LIN {X 0,Y 322.376,Z 758.442,A -85,B 0,C 180,E1 13709.907,E2 13709.907} C_VEL
LIN {X 0,Y 327.986,Z 742.44,A -85,B 0,C 180,E1 13707.682,E2 13707.682} C_VEL
LIN {X 0,Y 333.329,Z 725.588,A -85,B 0,C 180,E1 13705.781,E2 13705.781} C_VEL
LIN {X 0,Y 338.292,Z 707.747,A -85,B 0,C 180,E1 13704.157,E2 13704.157} C_VEL
LIN {X 0,Y 342.895,Z 688.344,A -85,B 0,C 180,E1 13702.762,E2 13702.762} C_VEL
LIN {X 0,Y 346.893,Z 667.6,A -85,B 0,C 180,E1 13701.623,E2 13701.623} C_VEL
LIN {X 0,Y 350,Z 646.538,A -85,B 0,C 180,E1 13700.791,E2 13700.791} C_VEL
LIN {X 0,Y 352.547,Z 620.24,A -85,B 0,C 180,E1 13700.102,E2 13700.102} C_VEL
LIN {X 0,Y 365.107,Z 463.823,A -85,B 0,C 180,E1 13696.583,E2 13696.583} C_VEL
LIN {X 0,Y 364.004,Z 412.304,A -85,B 0,C 180,E1 13693.947,E2 13693.947} C_VEL
LIN {X 0,Y 363.272,Z 382.468,A -85,B 0,C 180,E1 13692.235,E2 13692.235} C_VEL
LIN {X 0,Y 360.522,Z 376.636,A -85,B 0,C 180,E1 13690.87,E2 13690.87} C_VEL
LIN {X 0,Y 357.367,Z 367.476,A -85,B 0,C 180,E1 13688.041,E2 13688.041} C_VEL
LIN {X 0,Y 354.327,Z 359.067,A -85,B 0,C 180,E1 13684.856,E2 13684.856} C_VEL
LIN {X 0,Y 352.321,Z 354.194,A -85,B 0,C 180,E1 13682.439,E2 13682.439} C_VEL
LIN {X 0,Y 351.131,Z 351.132,A -85,B 0,C 180,E1 13680.652,E2 13680.652} C_VEL
LIN {X 0,Y 350.069,Z 347.943,A -85,B 0,C 180,E1 13678.363,E2 13678.363} C_VEL
LIN {X 0,Y 348.93,Z 344.03,A -85,B 0,C 180,E1 13673.583,E2 13673.583} C_VEL
LIN {X 0,Y 349.355,Z 344.256,A -85,B 0,C 180,E1 13668.944,E2 13668.944} C_VEL
LIN {X 0,Y 351.588,Z 349.237,A -85,B 0,C 180,E1 13663.817,E2 13663.817} C_VEL
LIN {X 0,Y 353.437,Z 352.672,A -85,B 0,C 180,E1 13661.698,E2 13661.698} C_VEL
LIN {X 0,Y 358.022,Z 358.691,A -85,B 0,C 180,E1 13659.226,E2 13659.226} C_VEL
LIN {X 0,Y 362.84,Z 365.211,A -85,B 0,C 180,E1 13657.05,E2 13657.05} C_VEL
LIN {X 0,Y 369.826,Z 375.683,A -85,B 0,C 180,E1 13654.369,E2 13654.369} C_VEL
LIN {X 0,Y 374.027,Z 382.841,A -85,B 0,C 180,E1 13652.929,E2 13652.929} C_VEL
LIN {X 0,Y 364.112,Z 552.249,A -85,B 0,C 180,E1 13649.475,E2 13649.475} C_VEL
LIN {X 0,Y 358.709,Z 656.095,A -85,B 0,C 180,E1 13647.399,E2 13647.399} C_VEL
LIN {X 0,Y 356.14,Z 678.482,A -85,B 0,C 180,E1 13646.754,E2 13646.754} C_VEL
LIN {X 0,Y 352.594,Z 700.34,A -85,B 0,C 180,E1 13645.893,E2 13645.893} C_VEL
LIN {X 0,Y 348.351,Z 721.516,A -85,B 0,C 180,E1 13644.793,E2 13644.793} C_VEL
LIN {X 0,Y 343.457,Z 741.511,A -85,B 0,C 180,E1 13643.46,E2 13643.46} C_VEL
LIN {X 0,Y 337.812,Z 761.919,A -85,B 0,C 180,E1 13641.786,E2 13641.786} C_VEL
LIN {X 0,Y 331.997,Z 780.753,A -85,B 0,C 180,E1 13639.9,E2 13639.9} C_VEL
LIN {X 0,Y 325.618,Z 799.71,A -85,B 0,C 180,E1 13637.599,E2 13637.599} C_VEL
LIN {X 0,Y 319.339,Z 817.406,A -85,B 0,C 180,E1 13635.038,E2 13635.038} C_VEL
LIN {X 0,Y 313.159,Z 834.22,A -85,B 0,C 180,E1 13632.102,E2 13632.102} C_VEL
LIN {X 0,Y 307.081,Z 850.603,A -85,B 0,C 180,E1 13628.69,E2 13628.69} C_VEL
LIN {X 0,Y 301.905,Z 865.076,A -85,B 0,C 180,E1 13625.112,E2 13625.112} C_VEL
LIN {X 0,Y 297.411,Z 878.3,A -85,B 0,C 180,E1 13621.177,E2 13621.177} C_VEL
LIN {X 0,Y 293.801,Z 890.287,A -85,B 0,C 180,E1 13616.909,E2 13616.909} C_VEL
LIN {X 0,Y 291.315,Z 900.346,A -85,B 0,C 180,E1 13612.605,E2 13612.605} C_VEL
LIN {X 0,Y 289.82,Z 908.415,A -85,B 0,C 180,E1 13608.295,E2 13608.295} C_VEL
LIN {X 0,Y 289.1,Z 914.862,A -85,B 0,C 180,E1 13604.008,E2 13604.008} C_VEL
LIN {X 0,Y 288.923,Z 919.155,A -85,B 0,C 180,E1 13600.163,E2 13600.163} C_VEL
LIN {X 0,Y 289.025,Z 922.186,A -85,B 0,C 180,E1 13596.354,E2 13596.354} C_VEL
LIN {X 0,Y 289.148,Z 923.885,A -85,B 0,C 180,E1 13592.376,E2 13592.376} C_VEL
LIN {X 0,Y 289.163,Z 924.136,A -85,B 0,C 180,E1 13589.007,E2 13589.007} C_VEL
LIN {X 0,Y 289.07,Z 923.328,A -85,B 0,C 180,E1 13585.634,E2 13585.634} C_VEL
LIN {X 0,Y 288.916,Z 921.176,A -85,B 0,C 180,E1 13581.798,E2 13581.798} C_VEL
LIN {X 0,Y 288.954,Z 917.176,A -85,B 0,C 180,E1 13577.61,E2 13577.61} C_VEL
LIN {X 0,Y 289.353,Z 912.158,A -85,B 0,C 180,E1 13573.744,E2 13573.744} C_VEL
LIN {X 0,Y 290.48,Z 904.897,A -85,B 0,C 180,E1 13569.432,E2 13569.432} C_VEL
LIN {X 0,Y 292.375,Z 896.411,A -85,B 0,C 180,E1 13565.339,E2 13565.339} C_VEL
LIN {X 0,Y 295.239,Z 886.029,A -85,B 0,C 180,E1 13561.254,E2 13561.254} C_VEL
LIN {X 0,Y 298.941,Z 874.449,A -85,B 0,C 180,E1 13557.417,E2 13557.417} C_VEL
LIN {X 0,Y 303.355,Z 861.486,A -85,B 0,C 180,E1 13553.842,E2 13553.842} C_VEL
LIN {X 0,Y 309.063,Z 845.63,A -85,B 0,C 180,E1 13550.165,E2 13550.165} C_VEL
LIN {X 0,Y 314.851,Z 829.645,A -85,B 0,C 180,E1 13547.062,E2 13547.062} C_VEL
LIN {X 0,Y 320.804,Z 812.678,A -85,B 0,C 180,E1 13544.331,E2 13544.331} C_VEL
LIN {X 0,Y 327.159,Z 793.761,A -85,B 0,C 180,E1 13541.778,E2 13541.778} C_VEL
LIN {X 0,Y 333.113,Z 774.835,A -85,B 0,C 180,E1 13539.653,E2 13539.653} C_VEL
LIN {X 0,Y 338.667,Z 754.972,A -85,B 0,C 180,E1 13537.836,E2 13537.836} C_VEL
LIN {X 0,Y 344.127,Z 733.064,A -85,B 0,C 180,E1 13536.208,E2 13536.208} C_VEL
LIN {X 0,Y 348.613,Z 712.087,A -85,B 0,C 180,E1 13534.964,E2 13534.964} C_VEL
LIN {X 0,Y 352.338,Z 690.211,A -85,B 0,C 180,E1 13533.974,E2 13533.974} C_VEL
LIN {X 0,Y 355.448,Z 666.338,A -85,B 0,C 180,E1 13533.189,E2 13533.189} C_VEL
LIN {X 0,Y 357.156,Z 643.717,A -85,B 0,C 180,E1 13532.651,E2 13532.651} C_VEL
LIN {X 0,Y 366.358,Z 456.176,A -85,B 0,C 180,E1 13528.938,E2 13528.938} C_VEL
LIN {X 0,Y 370.274,Z 382.007,A -85,B 0,C 180,E1 13527.414,E2 13527.414} C_VEL
LIN {X 0,Y 359.115,Z 365.438,A -85,B 0,C 180,E1 13524.51,E2 13524.51} C_VEL
LIN {X 0,Y 349.693,Z 352.331,A -85,B 0,C 180,E1 13521.821,E2 13521.821} C_VEL
LIN {X 0,Y 340.937,Z 340.666,A -85,B 0,C 180,E1 13518.998,E2 13518.998} C_VEL
LIN {X 0,Y 335.21,Z 330.431,A -85,B 0,C 180,E1 13515.573,E2 13515.573} C_VEL
LIN {X 0,Y 329.217,Z 320.51,A -85,B 0,C 180,E1 13511.564,E2 13511.564} C_VEL
LIN {X 0,Y 325.829,Z 315.067,A -85,B 0,C 180,E1 13509.004,E2 13509.004} C_VEL
LIN {X 0,Y 322.962,Z 310.321,A -85,B 0,C 180,E1 13506.578,E2 13506.578} C_VEL
LIN {X 0,Y 320.287,Z 306.211,A -85,B 0,C 180,E1 13504.118,E2 13504.118} C_VEL
LIN {X 0,Y 319.416,Z 304.812,A -85,B 0,C 180,E1 13503.231,E2 13503.231} C_VEL
LIN {X 0,Y 316.919,Z 301.182,A -85,B 0,C 180,E1 13500.543,E2 13500.543} C_VEL
LIN {X 0,Y 316.175,Z 299.504,A -85,B 0,C 180,E1 13499.457,E2 13499.457} C_VEL
LIN {X 0,Y 313.32,Z 295.951,A -85,B 0,C 180,E1 13495.792,E2 13495.792} C_VEL
LIN {X 0,Y 312.42,Z 293.809,A -85,B 0,C 180,E1 13493.938,E2 13493.938} C_VEL
LIN {X 0,Y 309.058,Z 289.36,A -85,B 0,C 180,E1 13485.385,E2 13485.385} C_VEL
LIN {X 0,Y 308.725,Z 288.453,A -85,B 0,C 180,E1 13481.3,E2 13481.3} C_VEL
LIN {X 0,Y 308.879,Z 289.021,A -85,B 0,C 180,E1 13477.143,E2 13477.143} C_VEL
LIN {X 0,Y 310.631,Z 292.387,A -85,B 0,C 180,E1 13470.285,E2 13470.285} C_VEL
LIN {X 0,Y 312.373,Z 294.134,A -85,B 0,C 180,E1 13467.253,E2 13467.253} C_VEL
LIN {X 0,Y 314.512,Z 298.285,A -85,B 0,C 180,E1 13463.525,E2 13463.525} C_VEL
LIN {X 0,Y 315.843,Z 299.683,A -85,B 0,C 180,E1 13462.025,E2 13462.025} C_VEL
LIN {X 0,Y 318.075,Z 303.861,A -85,B 0,C 180,E1 13459.169,E2 13459.169} C_VEL
LIN {X 0,Y 319.107,Z 305.22,A -85,B 0,C 180,E1 13458.135,E2 13458.135} C_VEL
LIN {X 0,Y 321.616,Z 309.49,A -85,B 0,C 180,E1 13455.615,E2 13455.615} C_VEL
LIN {X 0,Y 325.297,Z 315.942,A -85,B 0,C 180,E1 13452.311,E2 13452.311} C_VEL
LIN {X 0,Y 328.318,Z 321.379,A -85,B 0,C 180,E1 13449.877,E2 13449.877} C_VEL
LIN {X 0,Y 332.652,Z 329.233,A -85,B 0,C 180,E1 13446.738,E2 13446.738} C_VEL
LIN {X 0,Y 338.727,Z 341.166,A -85,B 0,C 180,E1 13442.728,E2 13442.728} C_VEL
LIN {X 0,Y 344.972,Z 354.709,A -85,B 0,C 180,E1 13438.921,E2 13438.921} C_VEL
LIN {X 0,Y 350.557,Z 368.131,A -85,B 0,C 180,E1 13435.694,E2 13435.694} C_VEL
LIN {X 0,Y 352.258,Z 372.767,A -85,B 0,C 180,E1 13434.703,E2 13434.703} C_VEL
LIN {X 0,Y 349.01,Z 389.794,A -85,B 0,C 180,E1 13433.272,E2 13433.272} C_VEL
LIN {X 0,Y 352.745,Z 460.829,A -85,B 0,C 180,E1 13429.925,E2 13429.925} C_VEL
LIN {X 0,Y 341.811,Z 627.739,A -85,B 0,C 180,E1 13426.223,E2 13426.223} C_VEL
LIN {X 0,Y 339.75,Z 649.403,A -85,B 0,C 180,E1 13425.59,E2 13425.59} C_VEL
LIN {X 0,Y 337.012,Z 669.497,A -85,B 0,C 180,E1 13424.723,E2 13424.723} C_VEL
LIN {X 0,Y 333.685,Z 688.632,A -85,B 0,C 180,E1 13423.606,E2 13423.606} C_VEL
LIN {X 0,Y 329.65,Z 707.702,A -85,B 0,C 180,E1 13422.171,E2 13422.171} C_VEL
LIN {X 0,Y 325.178,Z 725.794,A -85,B 0,C 180,E1 13420.454,E2 13420.454} C_VEL
LIN {X 0,Y 320.386,Z 742.938,A -85,B 0,C 180,E1 13418.436,E2 13418.436} C_VEL
LIN {X 0,Y 315.437,Z 759.06,A -85,B 0,C 180,E1 13416.097,E2 13416.097} C_VEL
LIN {X 0,Y 310.621,Z 773.611,A -85,B 0,C 180,E1 13413.508,E2 13413.508} C_VEL
LIN {X 0,Y 306.188,Z 786.321,A -85,B 0,C 180,E1 13410.75,E2 13410.75} C_VEL
LIN {X 0,Y 302.113,Z 797.741,A -85,B 0,C 180,E1 13407.726,E2 13407.726} C_VEL
LIN {X 0,Y 298.414,Z 808.119,A -85,B 0,C 180,E1 13404.325,E2 13404.325} C_VEL
LIN {X 0,Y 295.486,Z 816.535,A -85,B 0,C 180,E1 13400.851,E2 13400.851} C_VEL
LIN {X 0,Y 293.167,Z 823.725,A -85,B 0,C 180,E1 13396.994,E2 13396.994} C_VEL
LIN {X 0,Y 291.629,Z 829.062,A -85,B 0,C 180,E1 13393.046,E2 13393.046} C_VEL
LIN {X 0,Y 290.776,Z 832.595,A -85,B 0,C 180,E1 13389.049,E2 13389.049} C_VEL
LIN {X 0,Y 290.49,Z 834.354,A -85,B 0,C 180,E1 13385.173,E2 13385.173} C_VEL
LIN {X 0,Y 290.642,Z 834.535,A -85,B 0,C 180,E1 13381.309,E2 13381.309} C_VEL
LIN {X 0,Y 290.739,Z 834.351,A -85,B 0,C 180,E1 13380.486,E2 13380.486} C_VEL
LIN {X 0,Y 290.002,Z 834.043,A -85,B 0,C 180,E1 13378.964,E2 13378.964} C_VEL
LIN {X 0,Y 284.846,Z 832.664,A -85,B 0,C 180,E1 13374.855,E2 13374.855} C_VEL
LIN {X 0,Y 284.625,Z 831.626,A -85,B 0,C 180,E1 13373.525,E2 13373.525} C_VEL
LIN {X 0,Y 286.679,Z 826.967,A -85,B 0,C 180,E1 13369.558,E2 13369.558} C_VEL
LIN {X 0,Y 289.528,Z 820.722,A -85,B 0,C 180,E1 13365.77,E2 13365.77} C_VEL
LIN {X 0,Y 293.137,Z 813.011,A -85,B 0,C 180,E1 13362.216,E2 13362.216} C_VEL
LIN {X 0,Y 297.876,Z 802.822,A -85,B 0,C 180,E1 13358.551,E2 13358.551} C_VEL
LIN {X 0,Y 303.206,Z 791.159,A -85,B 0,C 180,E1 13355.244,E2 13355.244} C_VEL
LIN {X 0,Y 308.885,Z 778.138,A -85,B 0,C 180,E1 13352.282,E2 13352.282} C_VEL
LIN {X 0,Y 314.95,Z 763.342,A -85,B 0,C 180,E1 13349.563,E2 13349.563} C_VEL
LIN {X 0,Y 320.749,Z 747.985,A -85,B 0,C 180,E1 13347.272,E2 13347.272} C_VEL
LIN {X 0,Y 326.293,Z 731.895,A -85,B 0,C 180,E1 13345.321,E2 13345.321} C_VEL
LIN {X 0,Y 331.816,Z 713.67,A -85,B 0,C 180,E1 13343.533,E2 13343.533} C_VEL
LIN {X 0,Y 336.82,Z 694.445,A -85,B 0,C 180,E1 13342.046,E2 13342.046} C_VEL
LIN {X 0,Y 341.032,Z 674.694,A -85,B 0,C 180,E1 13340.866,E2 13340.866} C_VEL
LIN {X 0,Y 344.445,Z 654.269,A -85,B 0,C 180,E1 13339.961,E2 13339.961} C_VEL
LIN {X 0,Y 346.936,Z 633.468,A -85,B 0,C 180,E1 13339.325,E2 13339.325} C_VEL
LIN {X 0,Y 361.01,Z 465.78,A -85,B 0,C 180,E1 13335.544,E2 13335.544} C_VEL
LIN {X 0,Y 360.3,Z 414.273,A -85,B 0,C 180,E1 13332.867,E2 13332.867} C_VEL
LIN {X 0,Y 359.878,Z 387.613,A -85,B 0,C 180,E1 13331.336,E2 13331.336} C_VEL
LIN {X 0,Y 354.622,Z 377.047,A -85,B 0,C 180,E1 13328.634,E2 13328.634} C_VEL
LIN {X 0,Y 352.516,Z 371.95,A -85,B 0,C 180,E1 13327.005,E2 13327.005} C_VEL
LIN {X 0,Y 349.81,Z 364.508,A -85,B 0,C 180,E1 13323.933,E2 13323.933} C_VEL
LIN {X 0,Y 347.867,Z 358.86,A -85,B 0,C 180,E1 13320.988,E2 13320.988} C_VEL
LIN {X 0,Y 346.418,Z 354.914,A -85,B 0,C 180,E1 13318.015,E2 13318.015} C_VEL
LIN {X 0,Y 345.502,Z 351.238,A -85,B 0,C 180,E1 13313.352,E2 13313.352} C_VEL
LIN {X 0,Y 346.004,Z 351.513,A -85,B 0,C 180,E1 13309.005,E2 13309.005} C_VEL
LIN {X 0,Y 347.58,Z 355.306,A -85,B 0,C 180,E1 13304.995,E2 13304.995} C_VEL
LIN {X 0,Y 349.111,Z 357.114,A -85,B 0,C 180,E1 13303.785,E2 13303.785} C_VEL
LIN {X 0,Y 352.675,Z 361.524,A -85,B 0,C 180,E1 13301.486,E2 13301.486} C_VEL
LIN {X 0,Y 356.143,Z 366.162,A -85,B 0,C 180,E1 13299.584,E2 13299.584} C_VEL
LIN {X 0,Y 360.785,Z 372.607,A -85,B 0,C 180,E1 13297.428,E2 13297.428} C_VEL
LIN {X 0,Y 367.206,Z 382.565,A -85,B 0,C 180,E1 13294.864,E2 13294.864} C_VEL
LIN {X 0,Y 369.795,Z 387.109,A -85,B 0,C 180,E1 13293.918,E2 13293.918} C_VEL
LIN {X 0,Y 359.251,Z 558.947,A -85,B 0,C 180,E1 13290.394,E2 13290.394} C_VEL
LIN {X 0,Y 353.925,Z 655.866,A -85,B 0,C 180,E1 13288.437,E2 13288.437} C_VEL
LIN {X 0,Y 351.271,Z 678.222,A -85,B 0,C 180,E1 13287.793,E2 13287.793} C_VEL
LIN {X 0,Y 347.518,Z 700.481,A -85,B 0,C 180,E1 13286.91,E2 13286.91} C_VEL
LIN {X 0,Y 343.194,Z 721.167,A -85,B 0,C 180,E1 13285.829,E2 13285.829} C_VEL
LIN {X 0,Y 337.953,Z 741.723,A -85,B 0,C 180,E1 13284.446,E2 13284.446} C_VEL
LIN {X 0,Y 331.859,Z 762.75,A -85,B 0,C 180,E1 13282.69,E2 13282.69} C_VEL
LIN {X 0,Y 325.586,Z 782.198,A -85,B 0,C 180,E1 13280.7,E2 13280.7} C_VEL
LIN {X 0,Y 318.903,Z 800.994,A -85,B 0,C 180,E1 13278.341,E2 13278.341} C_VEL
LIN {X 0,Y 311.858,Z 819.725,A -85,B 0,C 180,E1 13275.506,E2 13275.506} C_VEL
LIN {X 0,Y 305.347,Z 836.674,A -85,B 0,C 180,E1 13272.416,E2 13272.416} C_VEL
LIN {X 0,Y 299.463,Z 851.692,A -85,B 0,C 180,E1 13269.124,E2 13269.124} C_VEL
LIN {X 0,Y 293.864,Z 866.497,A -85,B 0,C 180,E1 13265.255,E2 13265.255} C_VEL
LIN {X 0,Y 289.317,Z 879.444,A -85,B 0,C 180,E1 13261.221,E2 13261.221} C_VEL
LIN {X 0,Y 285.821,Z 890.486,A -85,B 0,C 180,E1 13257.047,E2 13257.047} C_VEL
LIN {X 0,Y 283.165,Z 900.845,A -85,B 0,C 180,E1 13252.312,E2 13252.312} C_VEL
LIN {X 0,Y 281.75,Z 908.514,A -85,B 0,C 180,E1 13247.981,E2 13247.981} C_VEL
LIN {X 0,Y 281.102,Z 914.575,A -85,B 0,C 180,E1 13243.575,E2 13243.575} C_VEL
LIN {X 0,Y 280.979,Z 918.672,A -85,B 0,C 180,E1 13239.626,E2 13239.626} C_VEL
LIN {X 0,Y 281.124,Z 921.527,A -85,B 0,C 180,E1 13235.508,E2 13235.508} C_VEL
LIN {X 0,Y 281.251,Z 922.767,A -85,B 0,C 180,E1 13231.831,E2 13231.831} C_VEL
LIN {X 0,Y 281.245,Z 922.851,A -85,B 0,C 180,E1 13228.368,E2 13228.368} C_VEL
LIN {X 0,Y 281.097,Z 921.712,A -85,B 0,C 180,E1 13224.487,E2 13224.487} C_VEL
LIN {X 0,Y 280.95,Z 918.889,A -85,B 0,C 180,E1 13220.334,E2 13220.334} C_VEL
LIN {X 0,Y 281.072,Z 914.947,A -85,B 0,C 180,E1 13216.419,E2 13216.419} C_VEL
LIN {X 0,Y 281.786,Z 908.587,A -85,B 0,C 180,E1 13211.803,E2 13211.803} C_VEL
LIN {X 0,Y 283.209,Z 901.186,A -85,B 0,C 180,E1 13207.584,E2 13207.584} C_VEL
LIN {X 0,Y 285.703,Z 891.494,A -85,B 0,C 180,E1 13203.161,E2 13203.161} C_VEL
LIN {X 0,Y 289.16,Z 880.465,A -85,B 0,C 180,E1 13198.986,E2 13198.986} C_VEL
LIN {X 0,Y 293.486,Z 867.988,A -85,B 0,C 180,E1 13195.084,E2 13195.084} C_VEL
LIN {X 0,Y 298.568,Z 854.204,A -85,B 0,C 180,E1 13191.471,E2 13191.471} C_VEL
LIN {X 0,Y 304.44,Z 838.727,A -85,B 0,C 180,E1 13188.059,E2 13188.059} C_VEL
LIN {X 0,Y 310.608,Z 822.164,A -85,B 0,C 180,E1 13185.041,E2 13185.041} C_VEL
LIN {X 0,Y 317.288,Z 803.6,A -85,B 0,C 180,E1 13182.22,E2 13182.22} C_VEL
LIN {X 0,Y 323.427,Z 785.574,A -85,B 0,C 180,E1 13179.941,E2 13179.941} C_VEL
LIN {X 0,Y 329.501,Z 765.926,A -85,B 0,C 180,E1 13177.91,E2 13177.91} C_VEL
LIN {X 0,Y 335.413,Z 744.664,A -85,B 0,C 180,E1 13176.112,E2 13176.112} C_VEL
LIN {X 0,Y 340.23,Z 724.92,A -85,B 0,C 180,E1 13174.759,E2 13174.759} C_VEL
LIN {X 0,Y 344.364,Z 704.453,A -85,B 0,C 180,E1 13173.654,E2 13173.654} C_VEL
LIN {X 0,Y 347.962,Z 682.722,A -85,B 0,C 180,E1 13172.749,E2 13172.749} C_VEL
LIN {X 0,Y 350.526,Z 660.938,A -85,B 0,C 180,E1 13172.092,E2 13172.092} C_VEL
LIN {X 0,Y 352.432,Z 629.266,A -85,B 0,C 180,E1 13171.41,E2 13171.41} C_VEL
LIN {X 0,Y 361.714,Z 449.353,A -85,B 0,C 180,E1 13167.813,E2 13167.813} C_VEL
LIN {X 0,Y 365.188,Z 386.033,A -85,B 0,C 180,E1 13166.506,E2 13166.506} C_VEL
LIN {X 0,Y 354.754,Z 370.415,A -85,B 0,C 180,E1 13163.681,E2 13163.681} C_VEL
LIN {X 0,Y 346.071,Z 358.262,A -85,B 0,C 180,E1 13161.127,E2 13161.127} C_VEL
LIN {X 0,Y 336.177,Z 345.236,A -85,B 0,C 180,E1 13157.895,E2 13157.895} C_VEL
LIN {X 0,Y 333.372,Z 341.225,A -85,B 0,C 180,E1 13156.734,E2 13156.734} C_VEL
LIN {X 0,Y 328.002,Z 331.87,A -85,B 0,C 180,E1 13153.217,E2 13153.217} C_VEL
LIN {X 0,Y 324.618,Z 326.4,A -85,B 0,C 180,E1 13150.83,E2 13150.83} C_VEL
LIN {X 0,Y 322.022,Z 321.96,A -85,B 0,C 180,E1 13148.752,E2 13148.752} C_VEL
LIN {X 0,Y 318.961,Z 316.989,A -85,B 0,C 180,E1 13146.119,E2 13146.119} C_VEL
LIN {X 0,Y 316.411,Z 312.7,A -85,B 0,C 180,E1 13143.624,E2 13143.624} C_VEL
LIN {X 0,Y 313.237,Z 308.01,A -85,B 0,C 180,E1 13140.184,E2 13140.184} C_VEL
LIN {X 0,Y 312.625,Z 306.631,A -85,B 0,C 180,E1 13139.268,E2 13139.268} C_VEL
LIN {X 0,Y 309.807,Z 303.026,A -85,B 0,C 180,E1 13135.558,E2 13135.558} C_VEL
LIN {X 0,Y 309.034,Z 301.05,A -85,B 0,C 180,E1 13133.872,E2 13133.872} C_VEL
LIN {X 0,Y 305.695,Z 296.575,A -85,B 0,C 180,E1 13125.22,E2 13125.22} C_VEL
LIN {X 0,Y 305.385,Z 295.716,A -85,B 0,C 180,E1 13121.127,E2 13121.127} C_VEL
LIN {X 0,Y 305.531,Z 296.396,A -85,B 0,C 180,E1 13116.868,E2 13116.868} C_VEL
LIN {X 0,Y 307.967,Z 300.334,A -85,B 0,C 180,E1 13108.922,E2 13108.922} C_VEL
LIN {X 0,Y 308.886,Z 301.457,A -85,B 0,C 180,E1 13107.278,E2 13107.278} C_VEL
LIN {X 0,Y 311.089,Z 305.568,A -85,B 0,C 180,E1 13103.469,E2 13103.469} C_VEL
LIN {X 0,Y 312.13,Z 306.647,A -85,B 0,C 180,E1 13102.279,E2 13102.279} C_VEL
LIN {X 0,Y 314.551,Z 311.094,A -85,B 0,C 180,E1 13099.161,E2 13099.161} C_VEL
LIN {X 0,Y 315.482,Z 312.618,A -85,B 0,C 180,E1 13098.143,E2 13098.143} C_VEL
LIN {X 0,Y 318.383,Z 317.548,A -85,B 0,C 180,E1 13095.215,E2 13095.215} C_VEL
LIN {X 0,Y 321.398,Z 322.978,A -85,B 0,C 180,E1 13092.462,E2 13092.462} C_VEL
LIN {X 0,Y 324.498,Z 328.674,A -85,B 0,C 180,E1 13089.896,E2 13089.896} C_VEL
LIN {X 0,Y 328.621,Z 336.388,A -85,B 0,C 180,E1 13086.828,E2 13086.828} C_VEL
LIN {X 0,Y 334.145,Z 347.38,A -85,B 0,C 180,E1 13083.089,E2 13083.089} C_VEL
LIN {X 0,Y 340.267,Z 360.945,A -85,B 0,C 180,E1 13079.226,E2 13079.226} C_VEL
LIN {X 0,Y 345.459,Z 373.779,A -85,B 0,C 180,E1 13076.101,E2 13076.101} C_VEL
LIN {X 0,Y 346.531,Z 376.658,A -85,B 0,C 180,E1 13075.464,E2 13075.464} C_VEL
LIN {X 0,Y 344.188,Z 388.923,A -85,B 0,C 180,E1 13074.438,E2 13074.438} C_VEL
LIN {X 0,Y 347.643,Z 461.101,A -85,B 0,C 180,E1 13070.968,E2 13070.968} C_VEL
LIN {X 0,Y 347.071,Z 472.125,A -85,B 0,C 180,E1 13070.692,E2 13070.692} C_VEL
LIN {X 0,Y 335.886,Z 634.097,A -85,B 0,C 180,E1 13067.063,E2 13067.063} C_VEL
LIN {X 0,Y 333.561,Z 655.179,A -85,B 0,C 180,E1 13066.367,E2 13066.367} C_VEL
LIN {X 0,Y 330.58,Z 674.831,A -85,B 0,C 180,E1 13065.438,E2 13065.438} C_VEL
LIN {X 0,Y 326.753,Z 694.856,A -85,B 0,C 180,E1 13064.172,E2 13064.172} C_VEL
LIN {X 0,Y 322.31,Z 714.147,A -85,B 0,C 180,E1 13062.596,E2 13062.596} C_VEL
LIN {X 0,Y 317.406,Z 732.447,A -85,B 0,C 180,E1 13060.713,E2 13060.713} C_VEL
LIN {X 0,Y 312.475,Z 748.885,A -85,B 0,C 180,E1 13058.615,E2 13058.615} C_VEL
LIN {X 0,Y 307.231,Z 764.847,A -85,B 0,C 180,E1 13056.11,E2 13056.11} C_VEL
LIN {X 0,Y 302.318,Z 778.832,A -85,B 0,C 180,E1 13053.415,E2 13053.415} C_VEL
LIN {X 0,Y 297.592,Z 791.659,A -85,B 0,C 180,E1 13050.387,E2 13050.387} C_VEL
LIN {X 0,Y 293.331,Z 803.012,A -85,B 0,C 180,E1 13047.071,E2 13047.071} C_VEL
LIN {X 0,Y 289.768,Z 812.582,A -85,B 0,C 180,E1 13043.583,E2 13043.583} C_VEL
LIN {X 0,Y 286.959,Z 820.411,A -85,B 0,C 180,E1 13039.969,E2 13039.969} C_VEL
LIN {X 0,Y 284.896,Z 826.671,A -85,B 0,C 180,E1 13036.195,E2 13036.195} C_VEL
LIN {X 0,Y 283.479,Z 831.489,A -85,B 0,C 180,E1 13032.132,E2 13032.132} C_VEL
LIN {X 0,Y 282.756,Z 834.554,A -85,B 0,C 180,E1 13027.989,E2 13027.989} C_VEL
LIN {X 0,Y 282.593,Z 835.843,A -85,B 0,C 180,E1 13023.98,E2 13023.98} C_VEL
LIN {X 0,Y 282.901,Z 835.524,A -85,B 0,C 180,E1 13019.984,E2 13019.984} C_VEL
LIN {X 0,Y 283.698,Z 833.722,A -85,B 0,C 180,E1 13016.165,E2 13016.165} C_VEL
LIN {X 0,Y 284.625,Z 831.626,A -85,B 0,C 180,E1 13013.525,E2 13013.525} C_VEL
LIN {X 0,Y 284.364,Z 830.337,A -85,B 0,C 180,E1 13011.984,E2 13011.984} C_VEL
LIN {X 0,Y 280.746,Z 826.443,A -85,B 0,C 180,E1 13007.924,E2 13007.924} C_VEL
LIN {X 0,Y 280.983,Z 824.416,A -85,B 0,C 180,E1 13006.51,E2 13006.51} C_VEL
LIN {X 0,Y 284.849,Z 816.657,A -85,B 0,C 180,E1 13002.516,E2 13002.516} C_VEL
LIN {X 0,Y 289.626,Z 807.031,A -85,B 0,C 180,E1 12998.725,E2 12998.725} C_VEL
LIN {X 0,Y 295.092,Z 795.788,A -85,B 0,C 180,E1 12995.261,E2 12995.261} C_VEL
LIN {X 0,Y 301.117,Z 782.883,A -85,B 0,C 180,E1 12992.091,E2 12992.091} C_VEL
LIN {X 0,Y 307.288,Z 768.795,A -85,B 0,C 180,E1 12989.311,E2 12989.311} C_VEL
LIN {X 0,Y 313.237,Z 754.082,A -85,B 0,C 180,E1 12986.952,E2 12986.952} C_VEL
LIN {X 0,Y 319.342,Z 737.61,A -85,B 0,C 180,E1 12984.805,E2 12984.805} C_VEL
LIN {X 0,Y 325.135,Z 719.962,A -85,B 0,C 180,E1 12982.952,E2 12982.952} C_VEL
LIN {X 0,Y 330.429,Z 701.288,A -85,B 0,C 180,E1 12981.391,E2 12981.391} C_VEL
LIN {X 0,Y 335.116,Z 681.624,A -85,B 0,C 180,E1 12980.107,E2 12980.107} C_VEL
LIN {X 0,Y 338.908,Z 661.79,A -85,B 0,C 180,E1 12979.128,E2 12979.128} C_VEL
LIN {X 0,Y 341.858,Z 641.111,A -85,B 0,C 180,E1 12978.399,E2 12978.399} C_VEL
LIN {X 0,Y 354.234,Z 500.386,A -85,B 0,C 180,E1 12975.178,E2 12975.178} C_VEL
LIN {X 0,Y 357.076,Z 466.271,A -85,B 0,C 180,E1 12974.403,E2 12974.403} C_VEL
LIN {X 0,Y 356.746,Z 414.625,A -85,B 0,C 180,E1 12971.672,E2 12971.672} C_VEL
LIN {X 0,Y 356.557,Z 392.616,A -85,B 0,C 180,E1 12970.379,E2 12970.379} C_VEL
LIN {X 0,Y 351.105,Z 381.373,A -85,B 0,C 180,E1 12967.321,E2 12967.321} C_VEL
LIN {X 0,Y 346.567,Z 372.275,A -85,B 0,C 180,E1 12964.053,E2 12964.053} C_VEL
LIN {X 0,Y 344.758,Z 367.804,A -85,B 0,C 180,E1 12961.828,E2 12961.828} C_VEL
LIN {X 0,Y 343.737,Z 364.849,A -85,B 0,C 180,E1 12959.999,E2 12959.999} C_VEL
LIN {X 0,Y 342.868,Z 362.011,A -85,B 0,C 180,E1 12957.827,E2 12957.827} C_VEL
LIN {X 0,Y 342.14,Z 358.494,A -85,B 0,C 180,E1 12953.287,E2 12953.287} C_VEL
LIN {X 0,Y 342.658,Z 358.75,A -85,B 0,C 180,E1 12949.236,E2 12949.236} C_VEL
LIN {X 0,Y 347.37,Z 364.352,A -85,B 0,C 180,E1 12944.302,E2 12944.302} C_VEL
LIN {X 0,Y 351.002,Z 369.077,A -85,B 0,C 180,E1 12941.825,E2 12941.825} C_VEL
LIN {X 0,Y 354.367,Z 373.74,A -85,B 0,C 180,E1 12939.908,E2 12939.908} C_VEL
LIN {X 0,Y 358.746,Z 380.006,A -85,B 0,C 180,E1 12937.811,E2 12937.811} C_VEL
LIN {X 0,Y 364.622,Z 389.446,A -85,B 0,C 180,E1 12935.366,E2 12935.366} C_VEL
LIN {X 0,Y 365.722,Z 391.705,A -85,B 0,C 180,E1 12934.927,E2 12934.927} C_VEL
LIN {X 0,Y 355.012,Z 557.395,A -85,B 0,C 180,E1 12931.509,E2 12931.509} C_VEL
LIN {X 0,Y 349.331,Z 655.447,A -85,B 0,C 180,E1 12929.514,E2 12929.514} C_VEL
LIN {X 0,Y 346.575,Z 677.793,A -85,B 0,C 180,E1 12928.869,E2 12928.869} C_VEL
LIN {X 0,Y 342.739,Z 699.729,A -85,B 0,C 180,E1 12928.001,E2 12928.001} C_VEL
LIN {X 0,Y 338.129,Z 721.004,A -85,B 0,C 180,E1 12926.888,E2 12926.888} C_VEL
LIN {X 0,Y 332.85,Z 740.983,A -85,B 0,C 180,E1 12925.542,E2 12925.542} C_VEL
LIN {X 0,Y 326.463,Z 762.151,A -85,B 0,C 180,E1 12923.764,E2 12923.764} C_VEL
LIN {X 0,Y 320.008,Z 781.41,A -85,B 0,C 180,E1 12921.782,E2 12921.782} C_VEL
LIN {X 0,Y 313.162,Z 799.861,A -85,B 0,C 180,E1 12919.45,E2 12919.45} C_VEL
LIN {X 0,Y 305.707,Z 818.798,A -85,B 0,C 180,E1 12916.555,E2 12916.555} C_VEL
LIN {X 0,Y 298.971,Z 835.498,A -85,B 0,C 180,E1 12913.471,E2 12913.471} C_VEL
LIN {X 0,Y 292.528,Z 851.119,A -85,B 0,C 180,E1 12909.982,E2 12909.982} C_VEL
LIN {X 0,Y 286.73,Z 865.577,A -85,B 0,C 180,E1 12906.106,E2 12906.106} C_VEL
LIN {X 0,Y 281.845,Z 878.665,A -85,B 0,C 180,E1 12901.907,E2 12901.907} C_VEL
LIN {X 0,Y 278.15,Z 889.666,A -85,B 0,C 180,E1 12897.624,E2 12897.624} C_VEL
LIN {X 0,Y 275.375,Z 899.748,A -85,B 0,C 180,E1 12892.859,E2 12892.859} C_VEL
LIN {X 0,Y 273.834,Z 907.579,A -85,B 0,C 180,E1 12888.299,E2 12888.299} C_VEL
LIN {X 0,Y 273.158,Z 913.558,A -85,B 0,C 180,E1 12883.762,E2 12883.762} C_VEL
LIN {X 0,Y 273.038,Z 917.619,A -85,B 0,C 180,E1 12879.695,E2 12879.695} C_VEL
LIN {X 0,Y 273.21,Z 920.386,A -85,B 0,C 180,E1 12875.458,E2 12875.458} C_VEL
LIN {X 0,Y 273.343,Z 921.544,A -85,B 0,C 180,E1 12871.884,E2 12871.884} C_VEL
LIN {X 0,Y 273.341,Z 921.648,A -85,B 0,C 180,E1 12868.531,E2 12868.531} C_VEL
LIN {X 0,Y 273.195,Z 920.634,A -85,B 0,C 180,E1 12864.748,E2 12864.748} C_VEL
LIN {X 0,Y 273.017,Z 918.01,A -85,B 0,C 180,E1 12860.512,E2 12860.512} C_VEL
LIN {X 0,Y 273.1,Z 914.358,A -85,B 0,C 180,E1 12856.662,E2 12856.662} C_VEL
LIN {X 0,Y 273.72,Z 908.596,A -85,B 0,C 180,E1 12852.129,E2 12852.129} C_VEL
LIN {X 0,Y 275.103,Z 901.364,A -85,B 0,C 180,E1 12847.789,E2 12847.789} C_VEL
LIN {X 0,Y 277.723,Z 891.537,A -85,B 0,C 180,E1 12843.021,E2 12843.021} C_VEL
LIN {X 0,Y 281.258,Z 880.729,A -85,B 0,C 180,E1 12838.731,E2 12838.731} C_VEL
LIN {X 0,Y 285.696,Z 868.422,A -85,B 0,C 180,E1 12834.726,E2 12834.726} C_VEL
LIN {X 0,Y 291.241,Z 854.089,A -85,B 0,C 180,E1 12830.823,E2 12830.823} C_VEL
LIN {X 0,Y 297.144,Z 839.174,A -85,B 0,C 180,E1 12827.439,E2 12827.439} C_VEL
LIN {X 0,Y 303.506,Z 822.829,A -85,B 0,C 180,E1 12824.365,E2 12824.365} C_VEL
LIN {X 0,Y 310.157,Z 805.176,A -85,B 0,C 180,E1 12821.589,E2 12821.589} C_VEL
LIN {X 0,Y 316.446,Z 787.395,A -85,B 0,C 180,E1 12819.273,E2 12819.273} C_VEL
LIN {X 0,Y 322.904,Z 767.562,A -85,B 0,C 180,E1 12817.144,E2 12817.144} C_VEL
LIN {X 0,Y 328.734,Z 747.721,A -85,B 0,C 180,E1 12815.397,E2 12815.397} C_VEL
LIN {X 0,Y 333.619,Z 728.482,A -85,B 0,C 180,E1 12814.035,E2 12814.035} C_VEL
LIN {X 0,Y 338.378,Z 706.472,A -85,B 0,C 180,E1 12812.788,E2 12812.788} C_VEL
LIN {X 0,Y 342.021,Z 685.767,A -85,B 0,C 180,E1 12811.888,E2 12811.888} C_VEL
LIN {X 0,Y 344.868,Z 663.558,A -85,B 0,C 180,E1 12811.187,E2 12811.187} C_VEL
LIN {X 0,Y 346.669,Z 638.606,A -85,B 0,C 180,E1 12810.612,E2 12810.612} C_VEL
LIN {X 0,Y 356.613,Z 452.449,A -85,B 0,C 180,E1 12806.868,E2 12806.868} C_VEL
LIN {X 0,Y 360.177,Z 390.021,A -85,B 0,C 180,E1 12805.574,E2 12805.574} C_VEL
LIN {X 0,Y 349.793,Z 374.444,A -85,B 0,C 180,E1 12802.655,E2 12802.655} C_VEL
LIN {X 0,Y 339.74,Z 360.385,A -85,B 0,C 180,E1 12799.514,E2 12799.514} C_VEL
LIN {X 0,Y 330.13,Z 347.876,A -85,B 0,C 180,E1 12796.179,E2 12796.179} C_VEL
LIN {X 0,Y 326.635,Z 343.156,A -85,B 0,C 180,E1 12794.719,E2 12794.719} C_VEL
LIN {X 0,Y 321.272,Z 333.981,A -85,B 0,C 180,E1 12790.944,E2 12790.944} C_VEL
LIN {X 0,Y 317.969,Z 328.538,A -85,B 0,C 180,E1 12788.317,E2 12788.317} C_VEL
LIN {X 0,Y 315.389,Z 324.127,A -85,B 0,C 180,E1 12786.006,E2 12786.006} C_VEL
LIN {X 0,Y 312.69,Z 319.559,A -85,B 0,C 180,E1 12783.3,E2 12783.3} C_VEL
LIN {X 0,Y 309.678,Z 315.143,A -85,B 0,C 180,E1 12780.001,E2 12780.001} C_VEL
LIN {X 0,Y 309.009,Z 313.709,A -85,B 0,C 180,E1 12779.015,E2 12779.015} C_VEL
LIN {X 0,Y 306.206,Z 309.872,A -85,B 0,C 180,E1 12775.131,E2 12775.131} C_VEL
LIN {X 0,Y 305.525,Z 308.197,A -85,B 0,C 180,E1 12773.612,E2 12773.612} C_VEL
LIN {X 0,Y 302.309,Z 303.723,A -85,B 0,C 180,E1 12764.855,E2 12764.855} C_VEL
LIN {X 0,Y 302.045,Z 302.988,A -85,B 0,C 180,E1 12760.87,E2 12760.87} C_VEL
LIN {X 0,Y 302.197,Z 303.763,A -85,B 0,C 180,E1 12756.608,E2 12756.608} C_VEL
LIN {X 0,Y 305.25,Z 308.141,A -85,B 0,C 180,E1 12747.842,E2 12747.842} C_VEL
LIN {X 0,Y 307.439,Z 312.603,A -85,B 0,C 180,E1 12743.709,E2 12743.709} C_VEL
LIN {X 0,Y 308.466,Z 313.75,A -85,B 0,C 180,E1 12742.456,E2 12742.456} C_VEL
LIN {X 0,Y 310.926,Z 318.216,A -85,B 0,C 180,E1 12739.249,E2 12739.249} C_VEL
LIN {X 0,Y 314.557,Z 324.61,A -85,B 0,C 180,E1 12735.376,E2 12735.376} C_VEL
LIN {X 0,Y 317.332,Z 329.659,A -85,B 0,C 180,E1 12732.767,E2 12732.767} C_VEL
LIN {X 0,Y 320.425,Z 335.44,A -85,B 0,C 180,E1 12730.139,E2 12730.139} C_VEL
LIN {X 0,Y 324.739,Z 343.795,A -85,B 0,C 180,E1 12726.821,E2 12726.821} C_VEL
LIN {X 0,Y 329.815,Z 354.192,A -85,B 0,C 180,E1 12723.281,E2 12723.281} C_VEL
LIN {X 0,Y 335.567,Z 367.184,A -85,B 0,C 180,E1 12719.538,E2 12719.538} C_VEL
LIN {X 0,Y 340.816,Z 380.613,A -85,B 0,C 180,E1 12716.25,E2 12716.25} C_VEL
LIN {X 0,Y 339.456,Z 388.172,A -85,B 0,C 180,E1 12715.624,E2 12715.624} C_VEL
LIN {X 0,Y 342.48,Z 457.929,A -85,B 0,C 180,E1 12712.2,E2 12712.2} C_VEL
LIN {X 0,Y 342.619,Z 465.563,A -85,B 0,C 180,E1 12711.886,E2 12711.886} C_VEL
LIN {X 0,Y 330.68,Z 632.986,A -85,B 0,C 180,E1 12708.125,E2 12708.125} C_VEL
LIN {X 0,Y 328.243,Z 654.821,A -85,B 0,C 180,E1 12707.416,E2 12707.416} C_VEL
LIN {X 0,Y 325.035,Z 675.411,A -85,B 0,C 180,E1 12706.441,E2 12706.441} C_VEL
LIN {X 0,Y 321.073,Z 695.443,A -85,B 0,C 180,E1 12705.166,E2 12705.166} C_VEL
LIN {X 0,Y 316.563,Z 714.377,A -85,B 0,C 180,E1 12703.611,E2 12703.611} C_VEL
LIN {X 0,Y 311.405,Z 732.977,A -85,B 0,C 180,E1 12701.686,E2 12701.686} C_VEL
LIN {X 0,Y 306.166,Z 749.78,A -85,B 0,C 180,E1 12699.519,E2 12699.519} C_VEL
LIN {X 0,Y 300.717,Z 765.701,A -85,B 0,C 180,E1 12696.985,E2 12696.985} C_VEL
LIN {X 0,Y 295.623,Z 779.595,A -85,B 0,C 180,E1 12694.269,E2 12694.269} C_VEL
LIN {X 0,Y 290.661,Z 792.468,A -85,B 0,C 180,E1 12691.185,E2 12691.185} C_VEL
LIN {X 0,Y 286.165,Z 803.88,A -85,B 0,C 180,E1 12687.797,E2 12687.797} C_VEL
LIN {X 0,Y 282.389,Z 813.514,A -85,B 0,C 180,E1 12684.222,E2 12684.222} C_VEL
LIN {X 0,Y 279.406,Z 821.379,A -85,B 0,C 180,E1 12680.528,E2 12680.528} C_VEL
LIN {X 0,Y 277.196,Z 827.697,A -85,B 0,C 180,E1 12676.655,E2 12676.655} C_VEL
LIN {X 0,Y 275.666,Z 832.574,A -85,B 0,C 180,E1 12672.482,E2 12672.482} C_VEL
LIN {X 0,Y 274.877,Z 835.698,A -85,B 0,C 180,E1 12668.224,E2 12668.224} C_VEL
LIN {X 0,Y 274.686,Z 837.059,A -85,B 0,C 180,E1 12664.035,E2 12664.035} C_VEL
LIN {X 0,Y 275.009,Z 836.794,A -85,B 0,C 180,E1 12659.915,E2 12659.915} C_VEL
LIN {X 0,Y 275.902,Z 834.955,A -85,B 0,C 180,E1 12655.829,E2 12655.829} C_VEL
LIN {X 0,Y 277.561,Z 831.443,A -85,B 0,C 180,E1 12651.717,E2 12651.717} C_VEL
LIN {X 0,Y 280.132,Z 826.084,A -85,B 0,C 180,E1 12647.582,E2 12647.582} C_VEL
LIN {X 0,Y 280.983,Z 824.416,A -85,B 0,C 180,E1 12646.51,E2 12646.51} C_VEL
LIN {X 0,Y 281.34,Z 822.098,A -85,B 0,C 180,E1 12645,E2 12645} C_VEL
LIN {X 0,Y 279.54,Z 816.07,A -85,B 0,C 180,E1 12641.092,E2 12641.092} C_VEL
LIN {X 0,Y 280.34,Z 812.921,A -85,B 0,C 180,E1 12639.649,E2 12639.649} C_VEL
LIN {X 0,Y 285.727,Z 802.61,A -85,B 0,C 180,E1 12636.006,E2 12636.006} C_VEL
LIN {X 0,Y 291.913,Z 790.339,A -85,B 0,C 180,E1 12632.589,E2 12632.589} C_VEL
LIN {X 0,Y 298.601,Z 776.276,A -85,B 0,C 180,E1 12629.476,E2 12629.476} C_VEL
LIN {X 0,Y 305.222,Z 761.273,A -85,B 0,C 180,E1 12626.816,E2 12626.816} C_VEL
LIN {X 0,Y 311.598,Z 745.373,A -85,B 0,C 180,E1 12624.543,E2 12624.543} C_VEL
LIN {X 0,Y 317.748,Z 728.314,A -85,B 0,C 180,E1 12622.574,E2 12622.574} C_VEL
LIN {X 0,Y 323.483,Z 710.13,A -85,B 0,C 180,E1 12620.89,E2 12620.89} C_VEL
LIN {X 0,Y 328.727,Z 690.505,A -85,B 0,C 180,E1 12619.463,E2 12619.463} C_VEL
LIN {X 0,Y 333.192,Z 669.847,A -85,B 0,C 180,E1 12618.321,E2 12618.321} C_VEL
LIN {X 0,Y 336.703,Z 648.595,A -85,B 0,C 180,E1 12617.474,E2 12617.474} C_VEL
LIN {X 0,Y 339.317,Z 625.013,A -85,B 0,C 180,E1 12616.839,E2 12616.839} C_VEL
LIN {X 0,Y 353.309,Z 467.909,A -85,B 0,C 180,E1 12613.293,E2 12613.293} C_VEL
LIN {X 0,Y 353.406,Z 416.317,A -85,B 0,C 180,E1 12610.524,E2 12610.524} C_VEL
LIN {X 0,Y 353.389,Z 397.701,A -85,B 0,C 180,E1 12609.403,E2 12609.403} C_VEL
LIN {X 0,Y 348.637,Z 387.512,A -85,B 0,C 180,E1 12606.504,E2 12606.504} C_VEL
LIN {X 0,Y 344.776,Z 379.385,A -85,B 0,C 180,E1 12603.491,E2 12603.491} C_VEL
LIN {X 0,Y 342.53,Z 374.699,A -85,B 0,C 180,E1 12601.17,E2 12601.17} C_VEL
LIN {X 0,Y 340.95,Z 370.943,A -85,B 0,C 180,E1 12598.739,E2 12598.739} C_VEL
LIN {X 0,Y 340.297,Z 369.334,A -85,B 0,C 180,E1 12597.365,E2 12597.365} C_VEL
LIN {X 0,Y 339.973,Z 366.192,A -85,B 0,C 180,E1 12593.244,E2 12593.244} C_VEL
LIN {X 0,Y 341.624,Z 366.708,A -85,B 0,C 180,E1 12589.203,E2 12589.203} C_VEL
LIN {X 0,Y 345.945,Z 372.056,A -85,B 0,C 180,E1 12584.579,E2 12584.579} C_VEL
LIN {X 0,Y 349.341,Z 376.629,A -85,B 0,C 180,E1 12582.166,E2 12582.166} C_VEL
LIN {X 0,Y 352.547,Z 381.209,A -85,B 0,C 180,E1 12580.275,E2 12580.275} C_VEL
LIN {X 0,Y 356.805,Z 387.531,A -85,B 0,C 180,E1 12578.161,E2 12578.161} C_VEL
LIN {X 0,Y 361.833,Z 395.885,A -85,B 0,C 180,E1 12575.973,E2 12575.973} C_VEL
LIN {X 0,Y 350.433,Z 563.969,A -85,B 0,C 180,E1 12572.488,E2 12572.488} C_VEL
LIN {X 0,Y 344.871,Z 655.078,A -85,B 0,C 180,E1 12570.62,E2 12570.62} C_VEL
LIN {X 0,Y 341.996,Z 677.616,A -85,B 0,C 180,E1 12569.969,E2 12569.969} C_VEL
LIN {X 0,Y 338.114,Z 699.094,A -85,B 0,C 180,E1 12569.124,E2 12569.124} C_VEL
LIN {X 0,Y 333.479,Z 719.816,A -85,B 0,C 180,E1 12568.045,E2 12568.045} C_VEL
LIN {X 0,Y 327.877,Z 740.27,A -85,B 0,C 180,E1 12566.67,E2 12566.67} C_VEL
LIN {X 0,Y 321.333,Z 761.201,A -85,B 0,C 180,E1 12564.916,E2 12564.916} C_VEL
LIN {X 0,Y 314.586,Z 780.567,A -85,B 0,C 180,E1 12562.913,E2 12562.913} C_VEL
LIN {X 0,Y 307.444,Z 799.02,A -85,B 0,C 180,E1 12560.565,E2 12560.565} C_VEL
LIN {X 0,Y 299.908,Z 817.368,A -85,B 0,C 180,E1 12557.738,E2 12557.738} C_VEL
LIN {X 0,Y 292.713,Z 834.306,A -85,B 0,C 180,E1 12554.58,E2 12554.58} C_VEL
LIN {X 0,Y 286.016,Z 849.73,A -85,B 0,C 180,E1 12551.084,E2 12551.084} C_VEL
LIN {X 0,Y 279.849,Z 864.211,A -85,B 0,C 180,E1 12547.14,E2 12547.14} C_VEL
LIN {X 0,Y 274.873,Z 876.741,A -85,B 0,C 180,E1 12543.065,E2 12543.065} C_VEL
LIN {X 0,Y 270.677,Z 888.34,A -85,B 0,C 180,E1 12538.455,E2 12538.455} C_VEL
LIN {X 0,Y 267.666,Z 898.446,A -85,B 0,C 180,E1 12533.556,E2 12533.556} C_VEL
LIN {X 0,Y 265.981,Z 906.294,A -85,B 0,C 180,E1 12528.859,E2 12528.859} C_VEL
LIN {X 0,Y 265.233,Z 912.297,A -85,B 0,C 180,E1 12524.181,E2 12524.181} C_VEL
LIN {X 0,Y 265.096,Z 916.378,A -85,B 0,C 180,E1 12519.989,E2 12519.989} C_VEL
LIN {X 0,Y 265.288,Z 919.16,A -85,B 0,C 180,E1 12515.621,E2 12515.621} C_VEL
LIN {X 0,Y 265.433,Z 920.325,A -85,B 0,C 180,E1 12511.941,E2 12511.941} C_VEL
LIN {X 0,Y 265.433,Z 920.427,A -85,B 0,C 180,E1 12508.487,E2 12508.487} C_VEL
LIN {X 0,Y 265.273,Z 919.401,A -85,B 0,C 180,E1 12504.591,E2 12504.591} C_VEL
LIN {X 0,Y 265.077,Z 916.741,A -85,B 0,C 180,E1 12500.225,E2 12500.225} C_VEL
LIN {X 0,Y 265.177,Z 913.054,A -85,B 0,C 180,E1 12496.256,E2 12496.256} C_VEL
LIN {X 0,Y 265.866,Z 907.227,A -85,B 0,C 180,E1 12491.583,E2 12491.583} C_VEL
LIN {X 0,Y 267.372,Z 899.961,A -85,B 0,C 180,E1 12487.111,E2 12487.111} C_VEL
LIN {X 0,Y 270.243,Z 889.951,A -85,B 0,C 180,E1 12482.162,E2 12482.162} C_VEL
LIN {X 0,Y 274.005,Z 879.168,A -85,B 0,C 180,E1 12477.806,E2 12477.806} C_VEL
LIN {X 0,Y 278.748,Z 866.76,A -85,B 0,C 180,E1 12473.71,E2 12473.71} C_VEL
LIN {X 0,Y 284.792,Z 851.888,A -85,B 0,C 180,E1 12469.628,E2 12469.628} C_VEL
LIN {X 0,Y 291.153,Z 836.572,A -85,B 0,C 180,E1 12466.152,E2 12466.152} C_VEL
LIN {X 0,Y 297.823,Z 819.976,A -85,B 0,C 180,E1 12463.048,E2 12463.048} C_VEL
LIN {X 0,Y 304.848,Z 801.922,A -85,B 0,C 180,E1 12460.251,E2 12460.251} C_VEL
LIN {X 0,Y 311.347,Z 784.15,A -85,B 0,C 180,E1 12457.962,E2 12457.962} C_VEL
LIN {X 0,Y 317.561,Z 765.325,A -85,B 0,C 180,E1 12455.982,E2 12455.982} C_VEL
LIN {X 0,Y 323.839,Z 744.165,A -85,B 0,C 180,E1 12454.16,E2 12454.16} C_VEL
LIN {X 0,Y 328.911,Z 724.581,A -85,B 0,C 180,E1 12452.801,E2 12452.801} C_VEL
LIN {X 0,Y 333.433,Z 703.551,A -85,B 0,C 180,E1 12451.653,E2 12451.653} C_VEL
LIN {X 0,Y 337.192,Z 682.189,A -85,B 0,C 180,E1 12450.758,E2 12450.758} C_VEL
LIN {X 0,Y 339.908,Z 660.399,A -85,B 0,C 180,E1 12450.094,E2 12450.094} C_VEL
LIN {X 0,Y 341.933,Z 629.039,A -85,B 0,C 180,E1 12449.409,E2 12449.409} C_VEL
LIN {X 0,Y 351.923,Z 449.687,A -85,B 0,C 180,E1 12445.779,E2 12445.779} C_VEL
LIN {X 0,Y 355.244,Z 393.998,A -85,B 0,C 180,E1 12444.618,E2 12444.618} C_VEL
LIN {X 0,Y 344.8,Z 378.4,A -85,B 0,C 180,E1 12441.565,E2 12441.565} C_VEL
LIN {X 0,Y 334.622,Z 364.188,A -85,B 0,C 180,E1 12438.24,E2 12438.24} C_VEL
LIN {X 0,Y 326.452,Z 353.524,A -85,B 0,C 180,E1 12435.247,E2 12435.247} C_VEL
LIN {X 0,Y 320.058,Z 345.359,A -85,B 0,C 180,E1 12432.632,E2 12432.632} C_VEL
LIN {X 0,Y 316.282,Z 339.128,A -85,B 0,C 180,E1 12429.83,E2 12429.83} C_VEL
LIN {X 0,Y 313.92,Z 335.097,A -85,B 0,C 180,E1 12427.872,E2 12427.872} C_VEL
LIN {X 0,Y 311.434,Z 330.823,A -85,B 0,C 180,E1 12425.573,E2 12425.573} C_VEL
LIN {X 0,Y 308.545,Z 325.977,A -85,B 0,C 180,E1 12422.601,E2 12422.601} C_VEL
LIN {X 0,Y 305.973,Z 321.85,A -85,B 0,C 180,E1 12419.553,E2 12419.553} C_VEL
LIN {X 0,Y 305.325,Z 320.728,A -85,B 0,C 180,E1 12418.687,E2 12418.687} C_VEL
LIN {X 0,Y 302.627,Z 316.71,A -85,B 0,C 180,E1 12414.693,E2 12414.693} C_VEL
LIN {X 0,Y 302.01,Z 315.336,A -85,B 0,C 180,E1 12413.327,E2 12413.327} C_VEL
LIN {X 0,Y 298.95,Z 310.949,A -85,B 0,C 180,E1 12404.68,E2 12404.68} C_VEL
LIN {X 0,Y 298.706,Z 310.265,A -85,B 0,C 180,E1 12400.648,E2 12400.648} C_VEL
LIN {X 0,Y 298.851,Z 311.062,A -85,B 0,C 180,E1 12396.539,E2 12396.539} C_VEL
LIN {X 0,Y 301.741,Z 315.3,A -85,B 0,C 180,E1 12387.983,E2 12387.983} C_VEL
LIN {X 0,Y 303.995,Z 319.854,A -85,B 0,C 180,E1 12383.7,E2 12383.7} C_VEL
LIN {X 0,Y 304.869,Z 321.029,A -85,B 0,C 180,E1 12382.532,E2 12382.532} C_VEL
LIN {X 0,Y 307.473,Z 325.508,A -85,B 0,C 180,E1 12379.186,E2 12379.186} C_VEL
LIN {X 0,Y 310.678,Z 331.531,A -85,B 0,C 180,E1 12375.601,E2 12375.601} C_VEL
LIN {X 0,Y 313.322,Z 336.415,A -85,B 0,C 180,E1 12373.05,E2 12373.05} C_VEL
LIN {X 0,Y 317.346,Z 343.911,A -85,B 0,C 180,E1 12369.617,E2 12369.617} C_VEL
LIN {X 0,Y 322.108,Z 353.751,A -85,B 0,C 180,E1 12365.889,E2 12365.889} C_VEL
LIN {X 0,Y 326.782,Z 363.868,A -85,B 0,C 180,E1 12362.584,E2 12362.584} C_VEL
LIN {X 0,Y 332.21,Z 376.772,A -85,B 0,C 180,E1 12358.986,E2 12358.986} C_VEL
LIN {X 0,Y 335.138,Z 384.933,A -85,B 0,C 180,E1 12357.017,E2 12357.017} C_VEL
LIN {X 0,Y 334.937,Z 389.127,A -85,B 0,C 180,E1 12356.752,E2 12356.752} C_VEL
LIN {X 0,Y 337.628,Z 459.003,A -85,B 0,C 180,E1 12353.266,E2 12353.266} C_VEL
LIN {X 0,Y 337.735,Z 466.757,A -85,B 0,C 180,E1 12352.942,E2 12352.942} C_VEL
LIN {X 0,Y 325.401,Z 633.771,A -85,B 0,C 180,E1 12349.167,E2 12349.167} C_VEL
LIN {X 0,Y 322.9,Z 655.34,A -85,B 0,C 180,E1 12348.46,E2 12348.46} C_VEL
LIN {X 0,Y 319.585,Z 675.916,A -85,B 0,C 180,E1 12347.48,E2 12347.48} C_VEL
LIN {X 0,Y 315.455,Z 696.101,A -85,B 0,C 180,E1 12346.186,E2 12346.186} C_VEL
LIN {X 0,Y 310.812,Z 714.932,A -85,B 0,C 180,E1 12344.629,E2 12344.629} C_VEL
LIN {X 0,Y 305.652,Z 732.942,A -85,B 0,C 180,E1 12342.758,E2 12342.758} C_VEL
LIN {X 0,Y 299.94,Z 750.622,A -85,B 0,C 180,E1 12340.464,E2 12340.464} C_VEL
LIN {X 0,Y 294.274,Z 766.538,A -85,B 0,C 180,E1 12337.899,E2 12337.899} C_VEL
LIN {X 0,Y 288.65,Z 781.223,A -85,B 0,C 180,E1 12334.97,E2 12334.97} C_VEL
LIN {X 0,Y 283.487,Z 794.007,A -85,B 0,C 180,E1 12331.821,E2 12331.821} C_VEL
LIN {X 0,Y 278.8,Z 805.338,A -85,B 0,C 180,E1 12328.358,E2 12328.358} C_VEL
LIN {X 0,Y 274.736,Z 815.188,A -85,B 0,C 180,E1 12324.573,E2 12324.573} C_VEL
LIN {X 0,Y 271.556,Z 823.143,A -85,B 0,C 180,E1 12320.66,E2 12320.66} C_VEL
LIN {X 0,Y 269.262,Z 829.374,A -85,B 0,C 180,E1 12316.623,E2 12316.623} C_VEL
LIN {X 0,Y 267.797,Z 833.853,A -85,B 0,C 180,E1 12312.624,E2 12312.624} C_VEL
LIN {X 0,Y 266.973,Z 836.959,A -85,B 0,C 180,E1 12308.239,E2 12308.239} C_VEL
LIN {X 0,Y 266.782,Z 838.294,A -85,B 0,C 180,E1 12303.995,E2 12303.995} C_VEL
LIN {X 0,Y 267.118,Z 838.063,A -85,B 0,C 180,E1 12299.842,E2 12299.842} C_VEL
LIN {X 0,Y 268.039,Z 836.341,A -85,B 0,C 180,E1 12295.721,E2 12295.721} C_VEL
LIN {X 0,Y 269.905,Z 832.687,A -85,B 0,C 180,E1 12291.243,E2 12291.243} C_VEL
LIN {X 0,Y 272.661,Z 827.348,A -85,B 0,C 180,E1 12286.998,E2 12286.998} C_VEL
LIN {X 0,Y 276.307,Z 820.471,A -85,B 0,C 180,E1 12283.036,E2 12283.036} C_VEL
LIN {X 0,Y 280.34,Z 812.921,A -85,B 0,C 180,E1 12279.649,E2 12279.649} C_VEL
LIN {X 0,Y 281.289,Z 809.609,A -85,B 0,C 180,E1 12278.227,E2 12278.227} C_VEL
LIN {X 0,Y 281.209,Z 801.419,A -85,B 0,C 180,E1 12274.482,E2 12274.482} C_VEL
LIN {X 0,Y 282.592,Z 797.419,A -85,B 0,C 180,E1 12273.164,E2 12273.164} C_VEL
LIN {X 0,Y 289.388,Z 784.273,A -85,B 0,C 180,E1 12269.868,E2 12269.868} C_VEL
LIN {X 0,Y 296.266,Z 769.978,A -85,B 0,C 180,E1 12267.011,E2 12267.011} C_VEL
LIN {X 0,Y 303.208,Z 754.239,A -85,B 0,C 180,E1 12264.482,E2 12264.482} C_VEL
LIN {X 0,Y 309.66,Z 738.064,A -85,B 0,C 180,E1 12262.395,E2 12262.395} C_VEL
LIN {X 0,Y 315.805,Z 720.603,A -85,B 0,C 180,E1 12260.574,E2 12260.574} C_VEL
LIN {X 0,Y 321.503,Z 701.93,A -85,B 0,C 180,E1 12259.024,E2 12259.024} C_VEL
LIN {X 0,Y 326.497,Z 682.337,A -85,B 0,C 180,E1 12257.757,E2 12257.757} C_VEL
LIN {X 0,Y 330.531,Z 662.541,A -85,B 0,C 180,E1 12256.79,E2 12256.79} C_VEL
LIN {X 0,Y 333.676,Z 641.815,A -85,B 0,C 180,E1 12256.066,E2 12256.066} C_VEL
LIN {X 0,Y 347.55,Z 493.95,A -85,B 0,C 180,E1 12252.701,E2 12252.701} C_VEL
LIN {X 0,Y 349.751,Z 469.076,A -85,B 0,C 180,E1 12252.129,E2 12252.129} C_VEL
LIN {X 0,Y 350.276,Z 416.935,A -85,B 0,C 180,E1 12249.291,E2 12249.291} C_VEL
LIN {X 0,Y 350.377,Z 403.046,A -85,B 0,C 180,E1 12248.45,E2 12248.45} C_VEL
LIN {X 0,Y 346.351,Z 393.896,A -85,B 0,C 180,E1 12245.757,E2 12245.757} C_VEL
LIN {X 0,Y 342.854,Z 386.118,A -85,B 0,C 180,E1 12242.757,E2 12242.757} C_VEL
LIN {X 0,Y 340.579,Z 380.811,A -85,B 0,C 180,E1 12239.999,E2 12239.999} C_VEL
LIN {X 0,Y 339.263,Z 377.402,A -85,B 0,C 180,E1 12237.466,E2 12237.466} C_VEL
LIN {X 0,Y 338.928,Z 374.122,A -85,B 0,C 180,E1 12233.223,E2 12233.223} C_VEL
LIN {X 0,Y 340.484,Z 374.595,A -85,B 0,C 180,E1 12229.338,E2 12229.338} C_VEL
LIN {X 0,Y 344.527,Z 379.759,A -85,B 0,C 180,E1 12224.859,E2 12224.859} C_VEL
LIN {X 0,Y 347.695,Z 384.18,A -85,B 0,C 180,E1 12222.511,E2 12222.511} C_VEL
LIN {X 0,Y 350.883,Z 388.888,A -85,B 0,C 180,E1 12220.568,E2 12220.568} C_VEL
LIN {X 0,Y 355.114,Z 395.478,A -85,B 0,C 180,E1 12218.399,E2 12218.399} C_VEL
LIN {X 0,Y 358.059,Z 400.771,A -85,B 0,C 180,E1 12217.027,E2 12217.027} C_VEL
LIN {X 0,Y 346.485,Z 563.315,A -85,B 0,C 180,E1 12213.646,E2 12213.646} C_VEL
LIN {X 0,Y 340.592,Z 654.81,A -85,B 0,C 180,E1 12211.758,E2 12211.758} C_VEL
LIN {X 0,Y 337.631,Z 677.192,A -85,B 0,C 180,E1 12211.111,E2 12211.111} C_VEL
LIN {X 0,Y 333.569,Z 698.816,A -85,B 0,C 180,E1 12210.261,E2 12210.261} C_VEL
LIN {X 0,Y 328.829,Z 719.264,A -85,B 0,C 180,E1 12209.198,E2 12209.198} C_VEL
LIN {X 0,Y 323.094,Z 739.542,A -85,B 0,C 180,E1 12207.84,E2 12207.84} C_VEL
LIN {X 0,Y 316.265,Z 760.533,A -85,B 0,C 180,E1 12206.079,E2 12206.079} C_VEL
LIN {X 0,Y 309.241,Z 779.912,A -85,B 0,C 180,E1 12204.066,E2 12204.066} C_VEL
LIN {X 0,Y 301.851,Z 798.226,A -85,B 0,C 180,E1 12201.721,E2 12201.721} C_VEL
LIN {X 0,Y 294.039,Z 816.437,A -85,B 0,C 180,E1 12198.884,E2 12198.884} C_VEL
LIN {X 0,Y 286.631,Z 833.039,A -85,B 0,C 180,E1 12195.76,E2 12195.76} C_VEL
LIN {X 0,Y 279.614,Z 848.363,A -85,B 0,C 180,E1 12192.238,E2 12192.238} C_VEL
LIN {X 0,Y 273.07,Z 862.868,A -85,B 0,C 180,E1 12188.225,E2 12188.225} C_VEL
LIN {X 0,Y 267.513,Z 875.997,A -85,B 0,C 180,E1 12183.839,E2 12183.839} C_VEL
LIN {X 0,Y 263.247,Z 887.023,A -85,B 0,C 180,E1 12179.335,E2 12179.335} C_VEL
LIN {X 0,Y 259.988,Z 897.155,A -85,B 0,C 180,E1 12174.292,E2 12174.292} C_VEL
LIN {X 0,Y 258.131,Z 905.017,A -85,B 0,C 180,E1 12169.455,E2 12169.455} C_VEL
LIN {X 0,Y 257.302,Z 911.043,A -85,B 0,C 180,E1 12164.624,E2 12164.624} C_VEL
LIN {X 0,Y 257.15,Z 915.14,A -85,B 0,C 180,E1 12160.301,E2 12160.301} C_VEL
LIN {X 0,Y 257.367,Z 917.931,A -85,B 0,C 180,E1 12155.795,E2 12155.795} C_VEL
LIN {X 0,Y 257.525,Z 919.1,A -85,B 0,C 180,E1 12152,E2 12152} C_VEL
LIN {X 0,Y 257.525,Z 919.198,A -85,B 0,C 180,E1 12148.44,E2 12148.44} C_VEL
LIN {X 0,Y 257.352,Z 918.161,A -85,B 0,C 180,E1 12144.424,E2 12144.424} C_VEL
LIN {X 0,Y 257.141,Z 915.457,A -85,B 0,C 180,E1 12139.92,E2 12139.92} C_VEL
LIN {X 0,Y 257.258,Z 911.744,A -85,B 0,C 180,E1 12135.824,E2 12135.824} C_VEL
LIN {X 0,Y 258.078,Z 905.516,A -85,B 0,C 180,E1 12130.771,E2 12130.771} C_VEL
LIN {X 0,Y 259.671,Z 898.544,A -85,B 0,C 180,E1 12126.391,E2 12126.391} C_VEL
LIN {X 0,Y 262.58,Z 889.046,A -85,B 0,C 180,E1 12121.575,E2 12121.575} C_VEL
LIN {X 0,Y 266.589,Z 878.177,A -85,B 0,C 180,E1 12117.053,E2 12117.053} C_VEL
LIN {X 0,Y 271.583,Z 865.775,A -85,B 0,C 180,E1 12112.857,E2 12112.857} C_VEL
LIN {X 0,Y 277.759,Z 851.279,A -85,B 0,C 180,E1 12108.793,E2 12108.793} C_VEL
LIN {X 0,Y 284.371,Z 836.054,A -85,B 0,C 180,E1 12105.255,E2 12105.255} C_VEL
LIN {X 0,Y 291.233,Z 819.676,A -85,B 0,C 180,E1 12102.133,E2 12102.133} C_VEL
LIN {X 0,Y 298.616,Z 801.382,A -85,B 0,C 180,E1 12099.26,E2 12099.26} C_VEL
LIN {X 0,Y 305.578,Z 782.962,A -85,B 0,C 180,E1 12096.87,E2 12096.87} C_VEL
LIN {X 0,Y 312.014,Z 764.065,A -85,B 0,C 180,E1 12094.877,E2 12094.877} C_VEL
LIN {X 0,Y 318.495,Z 742.774,A -85,B 0,C 180,E1 12093.047,E2 12093.047} C_VEL
LIN {X 0,Y 323.818,Z 722.666,A -85,B 0,C 180,E1 12091.663,E2 12091.663} C_VEL
LIN {X 0,Y 328.467,Z 701.186,A -85,B 0,C 180,E1 12090.517,E2 12090.517} C_VEL
LIN {X 0,Y 332.457,Z 678,A -85,B 0,C 180,E1 12089.59,E2 12089.59} C_VEL
LIN {X 0,Y 335.131,Z 655.777,A -85,B 0,C 180,E1 12088.942,E2 12088.942} C_VEL
LIN {X 0,Y 347.12,Z 450.927,A -85,B 0,C 180,E1 12084.743,E2 12084.743} C_VEL
LIN {X 0,Y 350.353,Z 398.126,A -85,B 0,C 180,E1 12083.637,E2 12083.637} C_VEL
LIN {X 0,Y 340.051,Z 382.529,A -85,B 0,C 180,E1 12080.482,E2 12080.482} C_VEL
LIN {X 0,Y 329.541,Z 367.903,A -85,B 0,C 180,E1 12076.889,E2 12076.889} C_VEL
LIN {X 0,Y 321.25,Z 357.088,A -85,B 0,C 180,E1 12073.683,E2 12073.683} C_VEL
LIN {X 0,Y 313.458,Z 347.435,A -85,B 0,C 180,E1 12070.244,E2 12070.244} C_VEL
LIN {X 0,Y 310.089,Z 341.958,A -85,B 0,C 180,E1 12067.597,E2 12067.597} C_VEL
LIN {X 0,Y 307.813,Z 337.901,A -85,B 0,C 180,E1 12065.406,E2 12065.406} C_VEL
LIN {X 0,Y 304.771,Z 332.882,A -85,B 0,C 180,E1 12062.257,E2 12062.257} C_VEL
LIN {X 0,Y 302.235,Z 328.472,A -85,B 0,C 180,E1 12059.053,E2 12059.053} C_VEL
LIN {X 0,Y 299.001,Z 323.297,A -85,B 0,C 180,E1 12054.051,E2 12054.051} C_VEL
LIN {X 0,Y 298.245,Z 322.299,A -85,B 0,C 180,E1 12052.682,E2 12052.682} C_VEL
LIN {X 0,Y 295.6,Z 318.18,A -85,B 0,C 180,E1 12044.502,E2 12044.502} C_VEL
LIN {X 0,Y 295.372,Z 317.544,A -85,B 0,C 180,E1 12040.421,E2 12040.421} C_VEL
LIN {X 0,Y 295.504,Z 318.363,A -85,B 0,C 180,E1 12036.469,E2 12036.469} C_VEL
LIN {X 0,Y 298.257,Z 322.625,A -85,B 0,C 180,E1 12028.013,E2 12028.013} C_VEL
LIN {X 0,Y 300.552,Z 327.103,A -85,B 0,C 180,E1 12023.691,E2 12023.691} C_VEL
LIN {X 0,Y 301.291,Z 328.306,A -85,B 0,C 180,E1 12022.607,E2 12022.607} C_VEL
LIN {X 0,Y 304.134,Z 333.494,A -85,B 0,C 180,E1 12018.84,E2 12018.84} C_VEL
LIN {X 0,Y 306.849,Z 338.543,A -85,B 0,C 180,E1 12015.79,E2 12015.79} C_VEL
LIN {X 0,Y 309.417,Z 343.381,A -85,B 0,C 180,E1 12013.242,E2 12013.242} C_VEL
LIN {X 0,Y 313.124,Z 350.423,A -85,B 0,C 180,E1 12009.973,E2 12009.973} C_VEL
LIN {X 0,Y 317.66,Z 360.027,A -85,B 0,C 180,E1 12006.283,E2 12006.283} C_VEL
LIN {X 0,Y 322.292,Z 370.331,A -85,B 0,C 180,E1 12002.884,E2 12002.884} C_VEL
LIN {X 0,Y 327.379,Z 382.789,A -85,B 0,C 180,E1 11999.365,E2 11999.365} C_VEL
LIN {X 0,Y 329.117,Z 386.716,A -85,B 0,C 180,E1 11998.469,E2 11998.469} C_VEL
LIN {X 0,Y 330.533,Z 389.649,A -85,B 0,C 180,E1 11997.934,E2 11997.934} C_VEL
LIN {X 0,Y 332.814,Z 458.28,A -85,B 0,C 180,E1 11994.448,E2 11994.448} C_VEL
LIN {X 0,Y 332.967,Z 467.825,A -85,B 0,C 180,E1 11994.029,E2 11994.029} C_VEL
LIN {X 0,Y 320.3,Z 633.82,A -85,B 0,C 180,E1 11990.263,E2 11990.263} C_VEL
LIN {X 0,Y 317.705,Z 655.611,A -85,B 0,C 180,E1 11989.549,E2 11989.549} C_VEL
LIN {X 0,Y 314.243,Z 676.424,A -85,B 0,C 180,E1 11988.555,E2 11988.555} C_VEL
LIN {X 0,Y 310.004,Z 696.486,A -85,B 0,C 180,E1 11987.263,E2 11987.263} C_VEL
LIN {X 0,Y 305.161,Z 715.487,A -85,B 0,C 180,E1 11985.685,E2 11985.685} C_VEL
LIN {X 0,Y 299.808,Z 733.534,A -85,B 0,C 180,E1 11983.797,E2 11983.797} C_VEL
LIN {X 0,Y 294.096,Z 750.606,A -85,B 0,C 180,E1 11981.573,E2 11981.573} C_VEL
LIN {X 0,Y 288.187,Z 766.632,A -85,B 0,C 180,E1 11978.984,E2 11978.984} C_VEL
LIN {X 0,Y 282.438,Z 781.081,A -85,B 0,C 180,E1 11976.099,E2 11976.099} C_VEL
LIN {X 0,Y 276.978,Z 794.06,A -85,B 0,C 180,E1 11972.899,E2 11972.899} C_VEL
LIN {X 0,Y 272.265,Z 804.971,A -85,B 0,C 180,E1 11969.581,E2 11969.581} C_VEL
LIN {X 0,Y 268.084,Z 814.621,A -85,B 0,C 180,E1 11965.939,E2 11965.939} C_VEL
LIN {X 0,Y 264.555,Z 822.906,A -85,B 0,C 180,E1 11961.964,E2 11961.964} C_VEL
LIN {X 0,Y 261.846,Z 829.714,A -85,B 0,C 180,E1 11957.655,E2 11957.655} C_VEL
LIN {X 0,Y 260.055,Z 834.739,A -85,B 0,C 180,E1 11953.202,E2 11953.202} C_VEL
LIN {X 0,Y 259.153,Z 837.801,A -85,B 0,C 180,E1 11948.976,E2 11948.976} C_VEL
LIN {X 0,Y 258.866,Z 839.389,A -85,B 0,C 180,E1 11944.616,E2 11944.616} C_VEL
LIN {X 0,Y 259.176,Z 839.406,A -85,B 0,C 180,E1 11940.158,E2 11940.158} C_VEL
LIN {X 0,Y 260.176,Z 837.731,A -85,B 0,C 180,E1 11935.606,E2 11935.606} C_VEL
LIN {X 0,Y 261.996,Z 834.456,A -85,B 0,C 180,E1 11931.257,E2 11931.257} C_VEL
LIN {X 0,Y 264.636,Z 829.724,A -85,B 0,C 180,E1 11927.135,E2 11927.135} C_VEL
LIN {X 0,Y 268.406,Z 823.069,A -85,B 0,C 180,E1 11922.976,E2 11922.976} C_VEL
LIN {X 0,Y 273.397,Z 814.232,A -85,B 0,C 180,E1 11918.837,E2 11918.837} C_VEL
LIN {X 0,Y 279.154,Z 803.814,A -85,B 0,C 180,E1 11915.077,E2 11915.077} C_VEL
LIN {X 0,Y 282.592,Z 797.419,A -85,B 0,C 180,E1 11913.164,E2 11913.164} C_VEL
LIN {X 0,Y 284.083,Z 793.246,A -85,B 0,C 180,E1 11911.874,E2 11911.874} C_VEL
LIN {X 0,Y 285.42,Z 782.953,A -85,B 0,C 180,E1 11908.406,E2 11908.406} C_VEL
LIN {X 0,Y 287.226,Z 778.198,A -85,B 0,C 180,E1 11907.238,E2 11907.238} C_VEL
LIN {X 0,Y 294.511,Z 763.141,A -85,B 0,C 180,E1 11904.521,E2 11904.521} C_VEL
LIN {X 0,Y 301.496,Z 747.179,A -85,B 0,C 180,E1 11902.213,E2 11902.213} C_VEL
LIN {X 0,Y 308.026,Z 730.55,A -85,B 0,C 180,E1 11900.273,E2 11900.273} C_VEL
LIN {X 0,Y 314.36,Z 712.048,A -85,B 0,C 180,E1 11898.545,E2 11898.545} C_VEL
LIN {X 0,Y 320.089,Z 692.202,A -85,B 0,C 180,E1 11897.098,E2 11897.098} C_VEL
LIN {X 0,Y 324.925,Z 671.56,A -85,B 0,C 180,E1 11895.953,E2 11895.953} C_VEL
LIN {X 0,Y 328.61,Z 651.083,A -85,B 0,C 180,E1 11895.128,E2 11895.128} C_VEL
LIN {X 0,Y 331.292,Z 629.397,A -85,B 0,C 180,E1 11894.528,E2 11894.528} C_VEL
LIN {X 0,Y 346.377,Z 470.586,A -85,B 0,C 180,E1 11890.956,E2 11890.956} C_VEL
LIN {X 0,Y 347.332,Z 418.698,A -85,B 0,C 180,E1 11888.097,E2 11888.097} C_VEL
LIN {X 0,Y 347.516,Z 408.453,A -85,B 0,C 180,E1 11887.48,E2 11887.48} C_VEL
LIN {X 0,Y 344.23,Z 400.547,A -85,B 0,C 180,E1 11885.082,E2 11885.082} C_VEL
LIN {X 0,Y 341.144,Z 393.206,A -85,B 0,C 180,E1 11882.183,E2 11882.183} C_VEL
LIN {X 0,Y 339.054,Z 388.012,A -85,B 0,C 180,E1 11879.324,E2 11879.324} C_VEL
LIN {X 0,Y 338.069,Z 385.118,A -85,B 0,C 180,E1 11877.117,E2 11877.117} C_VEL
LIN {X 0,Y 337.917,Z 382.048,A -85,B 0,C 180,E1 11873.031,E2 11873.031} C_VEL
LIN {X 0,Y 339.346,Z 382.483,A -85,B 0,C 180,E1 11869.474,E2 11869.474} C_VEL
LIN {X 0,Y 343.118,Z 387.462,A -85,B 0,C 180,E1 11865.141,E2 11865.141} C_VEL
LIN {X 0,Y 346.067,Z 391.73,A -85,B 0,C 180,E1 11862.86,E2 11862.86} C_VEL
LIN {X 0,Y 349.258,Z 396.588,A -85,B 0,C 180,E1 11860.854,E2 11860.854} C_VEL
LIN {X 0,Y 353.669,Z 403.804,A -85,B 0,C 180,E1 11858.524,E2 11858.524} C_VEL
LIN {X 0,Y 354.492,Z 405.528,A -85,B 0,C 180,E1 11858.113,E2 11858.113} C_VEL
LIN {X 0,Y 342.216,Z 569.927,A -85,B 0,C 180,E1 11854.683,E2 11854.683} C_VEL
LIN {X 0,Y 336.493,Z 654.386,A -85,B 0,C 180,E1 11852.931,E2 11852.931} C_VEL
LIN {X 0,Y 333.422,Z 676.765,A -85,B 0,C 180,E1 11852.285,E2 11852.285} C_VEL
LIN {X 0,Y 329.248,Z 698.338,A -85,B 0,C 180,E1 11851.444,E2 11851.444} C_VEL
LIN {X 0,Y 324.326,Z 718.864,A -85,B 0,C 180,E1 11850.381,E2 11850.381} C_VEL
LIN {X 0,Y 318.185,Z 739.733,A -85,B 0,C 180,E1 11848.979,E2 11848.979} C_VEL
LIN {X 0,Y 311.353,Z 759.904,A -85,B 0,C 180,E1 11847.28,E2 11847.28} C_VEL
LIN {X 0,Y 304.103,Z 779.133,A -85,B 0,C 180,E1 11845.278,E2 11845.278} C_VEL
LIN {X 0,Y 296.391,Z 797.47,A -85,B 0,C 180,E1 11842.918,E2 11842.918} C_VEL
LIN {X 0,Y 288.223,Z 815.698,A -85,B 0,C 180,E1 11840.051,E2 11840.051} C_VEL
LIN {X 0,Y 280.558,Z 832.051,A -85,B 0,C 180,E1 11836.932,E2 11836.932} C_VEL
LIN {X 0,Y 273.32,Z 847.024,A -85,B 0,C 180,E1 11833.448,E2 11833.448} C_VEL
LIN {X 0,Y 266.389,Z 861.563,A -85,B 0,C 180,E1 11829.358,E2 11829.358} C_VEL
LIN {X 0,Y 260.722,Z 874.09,A -85,B 0,C 180,E1 11825.114,E2 11825.114} C_VEL
LIN {X 0,Y 255.886,Z 885.685,A -85,B 0,C 180,E1 11820.283,E2 11820.283} C_VEL
LIN {X 0,Y 252.343,Z 895.86,A -85,B 0,C 180,E1 11815.082,E2 11815.082} C_VEL
LIN {X 0,Y 250.302,Z 903.742,A -85,B 0,C 180,E1 11810.09,E2 11810.09} C_VEL
LIN {X 0,Y 249.372,Z 909.782,A -85,B 0,C 180,E1 11805.104,E2 11805.104} C_VEL
LIN {X 0,Y 249.201,Z 913.947,A -85,B 0,C 180,E1 11800.578,E2 11800.578} C_VEL
LIN {X 0,Y 249.438,Z 916.704,A -85,B 0,C 180,E1 11795.98,E2 11795.98} C_VEL
LIN {X 0,Y 249.614,Z 917.88,A -85,B 0,C 180,E1 11792.064,E2 11792.064} C_VEL
LIN {X 0,Y 249.617,Z 917.974,A -85,B 0,C 180,E1 11788.391,E2 11788.391} C_VEL
LIN {X 0,Y 249.432,Z 916.922,A -85,B 0,C 180,E1 11784.246,E2 11784.246} C_VEL
LIN {X 0,Y 249.199,Z 914.176,A -85,B 0,C 180,E1 11779.596,E2 11779.596} C_VEL
LIN {X 0,Y 249.334,Z 910.428,A -85,B 0,C 180,E1 11775.364,E2 11775.364} C_VEL
LIN {X 0,Y 250.187,Z 904.465,A -85,B 0,C 180,E1 11770.383,E2 11770.383} C_VEL
LIN {X 0,Y 252.006,Z 897.108,A -85,B 0,C 180,E1 11765.628,E2 11765.628} C_VEL
LIN {X 0,Y 255.162,Z 887.531,A -85,B 0,C 180,E1 11760.669,E2 11760.669} C_VEL
LIN {X 0,Y 259.468,Z 876.554,A -85,B 0,C 180,E1 11756.028,E2 11756.028} C_VEL
LIN {X 0,Y 264.785,Z 864.049,A -85,B 0,C 180,E1 11751.734,E2 11751.734} C_VEL
LIN {X 0,Y 271.347,Z 849.424,A -85,B 0,C 180,E1 11747.596,E2 11747.596} C_VEL
LIN {X 0,Y 278.003,Z 834.704,A -85,B 0,C 180,E1 11744.148,E2 11744.148} C_VEL
LIN {X 0,Y 285.275,Z 818.033,A -85,B 0,C 180,E1 11740.952,E2 11740.952} C_VEL
LIN {X 0,Y 292.85,Z 799.883,A -85,B 0,C 180,E1 11738.093,E2 11738.093} C_VEL
LIN {X 0,Y 299.955,Z 781.669,A -85,B 0,C 180,E1 11735.727,E2 11735.727} C_VEL
LIN {X 0,Y 306.58,Z 762.724,A -85,B 0,C 180,E1 11733.73,E2 11733.73} C_VEL
LIN {X 0,Y 312.959,Z 742.273,A -85,B 0,C 180,E1 11731.978,E2 11731.978} C_VEL
LIN {X 0,Y 318.536,Z 721.768,A -85,B 0,C 180,E1 11730.565,E2 11730.565} C_VEL
LIN {X 0,Y 323.214,Z 700.731,A -85,B 0,C 180,E1 11729.444,E2 11729.444} C_VEL
LIN {X 0,Y 327.306,Z 677.595,A -85,B 0,C 180,E1 11728.519,E2 11728.519} C_VEL
LIN {X 0,Y 330.047,Z 655.406,A -85,B 0,C 180,E1 11727.871,E2 11727.871} C_VEL
LIN {X 0,Y 342.598,Z 448.383,A -85,B 0,C 180,E1 11723.609,E2 11723.609} C_VEL
LIN {X 0,Y 345.539,Z 402.178,A -85,B 0,C 180,E1 11722.635,E2 11722.635} C_VEL
LIN {X 0,Y 334.89,Z 386.09,A -85,B 0,C 180,E1 11719.219,E2 11719.219} C_VEL
LIN {X 0,Y 325.131,Z 372.497,A -85,B 0,C 180,E1 11715.702,E2 11715.702} C_VEL
LIN {X 0,Y 317.728,Z 362.884,A -85,B 0,C 180,E1 11712.726,E2 11712.726} C_VEL
LIN {X 0,Y 311.223,Z 354.653,A -85,B 0,C 180,E1 11709.758,E2 11709.758} C_VEL
LIN {X 0,Y 306.122,Z 348.532,A -85,B 0,C 180,E1 11707.13,E2 11707.13} C_VEL
LIN {X 0,Y 303.827,Z 344.516,A -85,B 0,C 180,E1 11704.909,E2 11704.909} C_VEL
LIN {X 0,Y 301.158,Z 339.944,A -85,B 0,C 180,E1 11702.056,E2 11702.056} C_VEL
LIN {X 0,Y 298.682,Z 335.601,A -85,B 0,C 180,E1 11698.85,E2 11698.85} C_VEL
LIN {X 0,Y 295.528,Z 330.372,A -85,B 0,C 180,E1 11693.785,E2 11693.785} C_VEL
LIN {X 0,Y 293.733,Z 328.397,A -85,B 0,C 180,E1 11690.399,E2 11690.399} C_VEL
LIN {X 0,Y 292.217,Z 325.294,A -85,B 0,C 180,E1 11683.911,E2 11683.911} C_VEL
LIN {X 0,Y 292.021,Z 324.836,A -85,B 0,C 180,E1 11679.748,E2 11679.748} C_VEL
LIN {X 0,Y 292.204,Z 325.946,A -85,B 0,C 180,E1 11675.758,E2 11675.758} C_VEL
LIN {X 0,Y 294.785,Z 329.941,A -85,B 0,C 180,E1 11668.055,E2 11668.055} C_VEL
LIN {X 0,Y 297.106,Z 334.35,A -85,B 0,C 180,E1 11663.681,E2 11663.681} C_VEL
LIN {X 0,Y 300.251,Z 340.148,A -85,B 0,C 180,E1 11659.256,E2 11659.256} C_VEL
LIN {X 0,Y 303.004,Z 345.504,A -85,B 0,C 180,E1 11656.004,E2 11656.004} C_VEL
LIN {X 0,Y 305.545,Z 350.405,A -85,B 0,C 180,E1 11653.41,E2 11653.41} C_VEL
LIN {X 0,Y 309.031,Z 357.233,A -85,B 0,C 180,E1 11650.222,E2 11650.222} C_VEL
LIN {X 0,Y 313.454,Z 366.812,A -85,B 0,C 180,E1 11646.504,E2 11646.504} C_VEL
LIN {X 0,Y 317.813,Z 376.791,A -85,B 0,C 180,E1 11643.192,E2 11643.192} C_VEL
LIN {X 0,Y 321.182,Z 384.625,A -85,B 0,C 180,E1 11640.949,E2 11640.949} C_VEL
LIN {X 0,Y 326.353,Z 393.98,A -85,B 0,C 180,E1 11638.939,E2 11638.939} C_VEL
LIN {X 0,Y 328.306,Z 463.777,A -85,B 0,C 180,E1 11635.355,E2 11635.355} C_VEL
LIN {X 0,Y 328.244,Z 469.535,A -85,B 0,C 180,E1 11635.13,E2 11635.13} C_VEL
LIN {X 0,Y 315.205,Z 634.804,A -85,B 0,C 180,E1 11631.366,E2 11631.366} C_VEL
LIN {X 0,Y 312.545,Z 656.273,A -85,B 0,C 180,E1 11630.654,E2 11630.654} C_VEL
LIN {X 0,Y 309.008,Z 676.858,A -85,B 0,C 180,E1 11629.666,E2 11629.666} C_VEL
LIN {X 0,Y 304.628,Z 696.956,A -85,B 0,C 180,E1 11628.368,E2 11628.368} C_VEL
LIN {X 0,Y 299.613,Z 716.004,A -85,B 0,C 180,E1 11626.78,E2 11626.78} C_VEL
LIN {X 0,Y 293.817,Z 734.849,A -85,B 0,C 180,E1 11624.789,E2 11624.789} C_VEL
LIN {X 0,Y 287.754,Z 752.242,A -85,B 0,C 180,E1 11622.481,E2 11622.481} C_VEL
LIN {X 0,Y 281.548,Z 768.355,A -85,B 0,C 180,E1 11619.817,E2 11619.817} C_VEL
LIN {X 0,Y 275.581,Z 782.692,A -85,B 0,C 180,E1 11616.879,E2 11616.879} C_VEL
LIN {X 0,Y 269.901,Z 795.58,A -85,B 0,C 180,E1 11613.613,E2 11613.613} C_VEL
LIN {X 0,Y 264.703,Z 807.018,A -85,B 0,C 180,E1 11610.002,E2 11610.002} C_VEL
LIN {X 0,Y 260.38,Z 816.492,A -85,B 0,C 180,E1 11606.259,E2 11606.259} C_VEL
LIN {X 0,Y 256.74,Z 824.636,A -85,B 0,C 180,E1 11602.168,E2 11602.168} C_VEL
LIN {X 0,Y 253.954,Z 831.318,A -85,B 0,C 180,E1 11597.727,E2 11597.727} C_VEL
LIN {X 0,Y 252.136,Z 836.203,A -85,B 0,C 180,E1 11593.175,E2 11593.175} C_VEL
LIN {X 0,Y 251.194,Z 839.353,A -85,B 0,C 180,E1 11588.521,E2 11588.521} C_VEL
LIN {X 0,Y 250.97,Z 840.741,A -85,B 0,C 180,E1 11584.011,E2 11584.011} C_VEL
LIN {X 0,Y 251.342,Z 840.603,A -85,B 0,C 180,E1 11579.657,E2 11579.657} C_VEL
LIN {X 0,Y 252.45,Z 838.89,A -85,B 0,C 180,E1 11575.067,E2 11575.067} C_VEL
LIN {X 0,Y 254.507,Z 835.457,A -85,B 0,C 180,E1 11570.477,E2 11570.477} C_VEL
LIN {X 0,Y 257.597,Z 830.286,A -85,B 0,C 180,E1 11565.994,E2 11565.994} C_VEL
LIN {X 0,Y 261.649,Z 823.618,A -85,B 0,C 180,E1 11561.831,E2 11561.831} C_VEL
LIN {X 0,Y 266.83,Z 814.988,A -85,B 0,C 180,E1 11557.758,E2 11557.758} C_VEL
LIN {X 0,Y 272.96,Z 804.544,A -85,B 0,C 180,E1 11553.94,E2 11553.94} C_VEL
LIN {X 0,Y 279.816,Z 792.312,A -85,B 0,C 180,E1 11550.437,E2 11550.437} C_VEL
LIN {X 0,Y 287.226,Z 778.198,A -85,B 0,C 180,E1 11547.238,E2 11547.238} C_VEL
LIN {X 0,Y 289.103,Z 773.262,A -85,B 0,C 180,E1 11546.104,E2 11546.104} C_VEL
LIN {X 0,Y 291.42,Z 761.031,A -85,B 0,C 180,E1 11542.985,E2 11542.985} C_VEL
LIN {X 0,Y 293.418,Z 755.539,A -85,B 0,C 180,E1 11541.992,E2 11541.992} C_VEL
LIN {X 0,Y 300.742,Z 738.529,A -85,B 0,C 180,E1 11539.809,E2 11539.809} C_VEL
LIN {X 0,Y 307.394,Z 720.903,A -85,B 0,C 180,E1 11537.998,E2 11537.998} C_VEL
LIN {X 0,Y 313.411,Z 702.426,A -85,B 0,C 180,E1 11536.494,E2 11536.494} C_VEL
LIN {X 0,Y 318.813,Z 682.414,A -85,B 0,C 180,E1 11535.228,E2 11535.228} C_VEL
LIN {X 0,Y 323.133,Z 662.199,A -85,B 0,C 180,E1 11534.272,E2 11534.272} C_VEL
LIN {X 0,Y 326.404,Z 641.497,A -85,B 0,C 180,E1 11533.576,E2 11533.576} C_VEL
LIN {X 0,Y 341.003,Z 495.073,A -85,B 0,C 180,E1 11530.278,E2 11530.278} C_VEL
LIN {X 0,Y 343.192,Z 471.834,A -85,B 0,C 180,E1 11529.744,E2 11529.744} C_VEL
LIN {X 0,Y 344.61,Z 420.538,A -85,B 0,C 180,E1 11526.884,E2 11526.884} C_VEL
LIN {X 0,Y 344.773,Z 413.744,A -85,B 0,C 180,E1 11526.452,E2 11526.452} C_VEL
LIN {X 0,Y 342.006,Z 406.795,A -85,B 0,C 180,E1 11524.233,E2 11524.233} C_VEL
LIN {X 0,Y 339.413,Z 400.103,A -85,B 0,C 180,E1 11521.519,E2 11521.519} C_VEL
LIN {X 0,Y 337.712,Z 395.539,A -85,B 0,C 180,E1 11518.897,E2 11518.897} C_VEL
LIN {X 0,Y 336.909,Z 392.835,A -85,B 0,C 180,E1 11516.767,E2 11516.767} C_VEL
LIN {X 0,Y 336.872,Z 389.979,A -85,B 0,C 180,E1 11513.01,E2 11513.01} C_VEL
LIN {X 0,Y 338.305,Z 390.565,A -85,B 0,C 180,E1 11509.441,E2 11509.441} C_VEL
LIN {X 0,Y 341.808,Z 395.316,A -85,B 0,C 180,E1 11505.343,E2 11505.343} C_VEL
LIN {X 0,Y 344.568,Z 399.464,A -85,B 0,C 180,E1 11503.131,E2 11503.131} C_VEL
LIN {X 0,Y 348.214,Z 405.144,A -85,B 0,C 180,E1 11500.805,E2 11500.805} C_VEL
LIN {X 0,Y 351.063,Z 410.367,A -85,B 0,C 180,E1 11499.219,E2 11499.219} C_VEL
LIN {X 0,Y 338.449,Z 572.012,A -85,B 0,C 180,E1 11495.846,E2 11495.846} C_VEL
LIN {X 0,Y 332.556,Z 654.212,A -85,B 0,C 180,E1 11494.13,E2 11494.13} C_VEL
LIN {X 0,Y 329.408,Z 676.463,A -85,B 0,C 180,E1 11493.491,E2 11493.491} C_VEL
LIN {X 0,Y 325.038,Z 698.182,A -85,B 0,C 180,E1 11492.647,E2 11492.647} C_VEL
LIN {X 0,Y 319.969,Z 718.5,A -85,B 0,C 180,E1 11491.595,E2 11491.595} C_VEL
LIN {X 0,Y 313.827,Z 738.751,A -85,B 0,C 180,E1 11490.244,E2 11490.244} C_VEL
LIN {X 0,Y 306.616,Z 759.281,A -85,B 0,C 180,E1 11488.524,E2 11488.524} C_VEL
LIN {X 0,Y 299.084,Z 778.461,A -85,B 0,C 180,E1 11486.522,E2 11486.522} C_VEL
LIN {X 0,Y 291.074,Z 796.78,A -85,B 0,C 180,E1 11484.158,E2 11484.158} C_VEL
LIN {X 0,Y 282.565,Z 814.909,A -85,B 0,C 180,E1 11481.278,E2 11481.278} C_VEL
LIN {X 0,Y 274.802,Z 830.753,A -85,B 0,C 180,E1 11478.231,E2 11478.231} C_VEL
LIN {X 0,Y 266.748,Z 846.545,A -85,B 0,C 180,E1 11474.498,E2 11474.498} C_VEL
LIN {X 0,Y 259.488,Z 860.941,A -85,B 0,C 180,E1 11470.338,E2 11470.338} C_VEL
LIN {X 0,Y 253.214,Z 873.963,A -85,B 0,C 180,E1 11465.757,E2 11465.757} C_VEL
LIN {X 0,Y 248.291,Z 885.116,A -85,B 0,C 180,E1 11460.935,E2 11460.935} C_VEL
LIN {X 0,Y 244.6,Z 894.987,A -85,B 0,C 180,E1 11455.674,E2 11455.674} C_VEL
LIN {X 0,Y 242.425,Z 902.812,A -85,B 0,C 180,E1 11450.52,E2 11450.52} C_VEL
LIN {X 0,Y 241.452,Z 908.529,A -85,B 0,C 180,E1 11445.612,E2 11445.612} C_VEL
LIN {X 0,Y 241.252,Z 912.667,A -85,B 0,C 180,E1 11440.988,E2 11440.988} C_VEL
LIN {X 0,Y 241.499,Z 915.475,A -85,B 0,C 180,E1 11436.177,E2 11436.177} C_VEL
LIN {X 0,Y 241.694,Z 916.619,A -85,B 0,C 180,E1 11432.368,E2 11432.368} C_VEL
LIN {X 0,Y 241.715,Z 916.765,A -85,B 0,C 180,E1 11428.575,E2 11428.575} C_VEL
LIN {X 0,Y 241.53,Z 915.83,A -85,B 0,C 180,E1 11424.534,E2 11424.534} C_VEL
LIN {X 0,Y 241.27,Z 913.423,A -85,B 0,C 180,E1 11419.974,E2 11419.974} C_VEL
LIN {X 0,Y 241.379,Z 909.568,A -85,B 0,C 180,E1 11415.362,E2 11415.362} C_VEL
LIN {X 0,Y 242.239,Z 903.748,A -85,B 0,C 180,E1 11410.215,E2 11410.215} C_VEL
LIN {X 0,Y 244.126,Z 896.465,A -85,B 0,C 180,E1 11405.305,E2 11405.305} C_VEL
LIN {X 0,Y 247.602,Z 886.487,A -85,B 0,C 180,E1 11399.949,E2 11399.949} C_VEL
LIN {X 0,Y 252.19,Z 875.454,A -85,B 0,C 180,E1 11395.155,E2 11395.155} C_VEL
LIN {X 0,Y 257.768,Z 863.024,A -85,B 0,C 180,E1 11390.78,E2 11390.78} C_VEL
LIN {X 0,Y 264.262,Z 849.189,A -85,B 0,C 180,E1 11386.775,E2 11386.775} C_VEL
LIN {X 0,Y 271.388,Z 834.09,A -85,B 0,C 180,E1 11383.155,E2 11383.155} C_VEL
LIN {X 0,Y 278.965,Z 817.439,A -85,B 0,C 180,E1 11379.909,E2 11379.909} C_VEL
LIN {X 0,Y 286.792,Z 799.331,A -85,B 0,C 180,E1 11377.022,E2 11377.022} C_VEL
LIN {X 0,Y 294.113,Z 781.143,A -85,B 0,C 180,E1 11374.642,E2 11374.642} C_VEL
LIN {X 0,Y 301.056,Z 761.905,A -85,B 0,C 180,E1 11372.601,E2 11372.601} C_VEL
LIN {X 0,Y 307.537,Z 741.758,A -85,B 0,C 180,E1 11370.87,E2 11370.87} C_VEL
LIN {X 0,Y 313.07,Z 722.067,A -85,B 0,C 180,E1 11369.505,E2 11369.505} C_VEL
LIN {X 0,Y 317.926,Z 700.944,A -85,B 0,C 180,E1 11368.37,E2 11368.37} C_VEL
LIN {X 0,Y 322.147,Z 677.842,A -85,B 0,C 180,E1 11367.44,E2 11367.44} C_VEL
LIN {X 0,Y 324.994,Z 655.605,A -85,B 0,C 180,E1 11366.786,E2 11366.786} C_VEL
LIN {X 0,Y 337.941,Z 450.06,A -85,B 0,C 180,E1 11362.533,E2 11362.533} C_VEL
LIN {X 0,Y 340.812,Z 406.287,A -85,B 0,C 180,E1 11361.604,E2 11361.604} C_VEL
LIN {X 0,Y 331.15,Z 391.676,A -85,B 0,C 180,E1 11358.393,E2 11358.393} C_VEL
LIN {X 0,Y 321.915,Z 378.632,A -85,B 0,C 180,E1 11354.94,E2 11354.94} C_VEL
LIN {X 0,Y 314.943,Z 369.457,A -85,B 0,C 180,E1 11352.036,E2 11352.036} C_VEL
LIN {X 0,Y 308.546,Z 361.369,A -85,B 0,C 180,E1 11349.043,E2 11349.043} C_VEL
LIN {X 0,Y 303.4,Z 355.158,A -85,B 0,C 180,E1 11346.339,E2 11346.339} C_VEL
LIN {X 0,Y 299.916,Z 351.047,A -85,B 0,C 180,E1 11344.302,E2 11344.302} C_VEL
LIN {X 0,Y 297.433,Z 346.881,A -85,B 0,C 180,E1 11341.734,E2 11341.734} C_VEL
LIN {X 0,Y 294.674,Z 342.07,A -85,B 0,C 180,E1 11338.056,E2 11338.056} C_VEL
LIN {X 0,Y 292.042,Z 337.437,A -85,B 0,C 180,E1 11333.514,E2 11333.514} C_VEL
LIN {X 0,Y 288.991,Z 332.924,A -85,B 0,C 180,E1 11324.961,E2 11324.961} C_VEL
LIN {X 0,Y 288.711,Z 332.076,A -85,B 0,C 180,E1 11320.992,E2 11320.992} C_VEL
LIN {X 0,Y 288.783,Z 332.822,A -85,B 0,C 180,E1 11316.753,E2 11316.753} C_VEL
LIN {X 0,Y 291.253,Z 336.994,A -85,B 0,C 180,E1 11308.317,E2 11308.317} C_VEL
LIN {X 0,Y 293.534,Z 341.468,A -85,B 0,C 180,E1 11303.834,E2 11303.834} C_VEL
LIN {X 0,Y 296.56,Z 347.282,A -85,B 0,C 180,E1 11299.407,E2 11299.407} C_VEL
LIN {X 0,Y 298.976,Z 352.019,A -85,B 0,C 180,E1 11296.457,E2 11296.457} C_VEL
LIN {X 0,Y 301.68,Z 357.422,A -85,B 0,C 180,E1 11293.583,E2 11293.583} C_VEL
LIN {X 0,Y 304.938,Z 364.039,A -85,B 0,C 180,E1 11290.475,E2 11290.475} C_VEL
LIN {X 0,Y 308.998,Z 373.016,A -85,B 0,C 180,E1 11286.944,E2 11286.944} C_VEL
LIN {X 0,Y 313.155,Z 382.452,A -85,B 0,C 180,E1 11283.795,E2 11283.795} C_VEL
LIN {X 0,Y 320.546,Z 395.358,A -85,B 0,C 180,E1 11280.627,E2 11280.627} C_VEL
LIN {X 0,Y 322.241,Z 398.864,A -85,B 0,C 180,E1 11279.934,E2 11279.934} C_VEL
LIN {X 0,Y 323.851,Z 468.694,A -85,B 0,C 180,E1 11276.318,E2 11276.318} C_VEL
LIN {X 0,Y 310.301,Z 635.018,A -85,B 0,C 180,E1 11272.524,E2 11272.524} C_VEL
LIN {X 0,Y 307.555,Z 656.568,A -85,B 0,C 180,E1 11271.81,E2 11271.81} C_VEL
LIN {X 0,Y 303.892,Z 677.268,A -85,B 0,C 180,E1 11270.816,E2 11270.816} C_VEL
LIN {X 0,Y 299.367,Z 697.401,A -85,B 0,C 180,E1 11269.513,E2 11269.513} C_VEL
LIN {X 0,Y 294.175,Z 716.495,A -85,B 0,C 180,E1 11267.916,E2 11267.916} C_VEL
LIN {X 0,Y 288.168,Z 735.387,A -85,B 0,C 180,E1 11265.911,E2 11265.911} C_VEL
LIN {X 0,Y 281.808,Z 752.985,A -85,B 0,C 180,E1 11263.558,E2 11263.558} C_VEL
LIN {X 0,Y 275.4,Z 768.999,A -85,B 0,C 180,E1 11260.884,E2 11260.884} C_VEL
LIN {X 0,Y 269.164,Z 783.39,A -85,B 0,C 180,E1 11257.902,E2 11257.902} C_VEL
LIN {X 0,Y 263.21,Z 796.336,A -85,B 0,C 180,E1 11254.578,E2 11254.578} C_VEL
LIN {X 0,Y 257.737,Z 807.836,A -85,B 0,C 180,E1 11250.891,E2 11250.891} C_VEL
LIN {X 0,Y 253.167,Z 817.371,A -85,B 0,C 180,E1 11247.059,E2 11247.059} C_VEL
LIN {X 0,Y 249.297,Z 825.579,A -85,B 0,C 180,E1 11242.86,E2 11242.86} C_VEL
LIN {X 0,Y 246.313,Z 832.325,A -85,B 0,C 180,E1 11238.292,E2 11238.292} C_VEL
LIN {X 0,Y 244.354,Z 837.265,A -85,B 0,C 180,E1 11233.603,E2 11233.603} C_VEL
LIN {X 0,Y 243.321,Z 840.47,A -85,B 0,C 180,E1 11228.804,E2 11228.804} C_VEL
LIN {X 0,Y 243.061,Z 841.938,A -85,B 0,C 180,E1 11224.151,E2 11224.151} C_VEL
LIN {X 0,Y 243.45,Z 841.883,A -85,B 0,C 180,E1 11219.593,E2 11219.593} C_VEL
LIN {X 0,Y 244.634,Z 840.228,A -85,B 0,C 180,E1 11214.813,E2 11214.813} C_VEL
LIN {X 0,Y 246.751,Z 836.983,A -85,B 0,C 180,E1 11210.195,E2 11210.195} C_VEL
LIN {X 0,Y 249.852,Z 832.186,A -85,B 0,C 180,E1 11205.75,E2 11205.75} C_VEL
LIN {X 0,Y 254.222,Z 825.46,A -85,B 0,C 180,E1 11201.31,E2 11201.31} C_VEL
LIN {X 0,Y 259.619,Z 817.017,A -85,B 0,C 180,E1 11197.14,E2 11197.14} C_VEL
LIN {X 0,Y 265.869,Z 806.931,A -85,B 0,C 180,E1 11193.302,E2 11193.302} C_VEL
LIN {X 0,Y 272.524,Z 795.733,A -85,B 0,C 180,E1 11189.931,E2 11189.931} C_VEL
LIN {X 0,Y 279.635,Z 783.037,A -85,B 0,C 180,E1 11186.867,E2 11186.867} C_VEL
LIN {X 0,Y 287.25,Z 768.379,A -85,B 0,C 180,E1 11184.031,E2 11184.031} C_VEL
LIN {X 0,Y 293.418,Z 755.539,A -85,B 0,C 180,E1 11181.992,E2 11181.992} C_VEL
LIN {X 0,Y 295.447,Z 749.879,A -85,B 0,C 180,E1 11181.034,E2 11181.034} C_VEL
LIN {X 0,Y 298.32,Z 735.859,A -85,B 0,C 180,E1 11178.31,E2 11178.31} C_VEL
LIN {X 0,Y 300.257,Z 729.754,A -85,B 0,C 180,E1 11177.481,E2 11177.481} C_VEL
LIN {X 0,Y 306.651,Z 712.05,A -85,B 0,C 180,E1 11175.883,E2 11175.883} C_VEL
LIN {X 0,Y 312.646,Z 692.543,A -85,B 0,C 180,E1 11174.496,E2 11174.496} C_VEL
LIN {X 0,Y 317.775,Z 671.862,A -85,B 0,C 180,E1 11173.381,E2 11173.381} C_VEL
LIN {X 0,Y 321.727,Z 650.874,A -85,B 0,C 180,E1 11172.564,E2 11172.564} C_VEL
LIN {X 0,Y 324.587,Z 628.431,A -85,B 0,C 180,E1 11171.966,E2 11171.966} C_VEL
LIN {X 0,Y 340.247,Z 473.359,A -85,B 0,C 180,E1 11168.518,E2 11168.518} C_VEL
LIN {X 0,Y 342.09,Z 422.573,A -85,B 0,C 180,E1 11165.66,E2 11165.66} C_VEL
LIN {X 0,Y 342.152,Z 419.054,A -85,B 0,C 180,E1 11165.407,E2 11165.407} C_VEL
LIN {X 0,Y 339.38,Z 411.595,A -85,B 0,C 180,E1 11162.821,E2 11162.821} C_VEL
LIN {X 0,Y 337.42,Z 406.13,A -85,B 0,C 180,E1 11160.339,E2 11160.339} C_VEL
LIN {X 0,Y 336.281,Z 402.712,A -85,B 0,C 180,E1 11158.21,E2 11158.21} C_VEL
LIN {X 0,Y 335.798,Z 400.685,A -85,B 0,C 180,E1 11156.585,E2 11156.585} C_VEL
LIN {X 0,Y 335.865,Z 397.905,A -85,B 0,C 180,E1 11152.817,E2 11152.817} C_VEL
LIN {X 0,Y 337.165,Z 398.478,A -85,B 0,C 180,E1 11149.578,E2 11149.578} C_VEL
LIN {X 0,Y 340.414,Z 403.016,A -85,B 0,C 180,E1 11145.629,E2 11145.629} C_VEL
LIN {X 0,Y 342.992,Z 407.016,A -85,B 0,C 180,E1 11143.487,E2 11143.487} C_VEL
LIN {X 0,Y 346.393,Z 412.566,A -85,B 0,C 180,E1 11141.214,E2 11141.214} C_VEL
LIN {X 0,Y 347.834,Z 415.389,A -85,B 0,C 180,E1 11140.349,E2 11140.349} C_VEL
LIN {X 0,Y 334.76,Z 575.246,A -85,B 0,C 180,E1 11137.012,E2 11137.012} C_VEL
LIN {X 0,Y 328.861,Z 653.703,A -85,B 0,C 180,E1 11135.371,E2 11135.371} C_VEL
LIN {X 0,Y 325.577,Z 676.098,A -85,B 0,C 180,E1 11134.73,E2 11134.73} C_VEL
LIN {X 0,Y 320.98,Z 698.135,A -85,B 0,C 180,E1 11133.878,E2 11133.878} C_VEL
LIN {X 0,Y 315.769,Z 718.309,A -85,B 0,C 180,E1 11132.838,E2 11132.838} C_VEL
LIN {X 0,Y 309.445,Z 738.418,A -85,B 0,C 180,E1 11131.501,E2 11131.501} C_VEL
LIN {X 0,Y 301.936,Z 758.977,A -85,B 0,C 180,E1 11129.778,E2 11129.778} C_VEL
LIN {X 0,Y 294.201,Z 777.915,A -85,B 0,C 180,E1 11127.8,E2 11127.8} C_VEL
LIN {X 0,Y 285.933,Z 796.051,A -85,B 0,C 180,E1 11125.45,E2 11125.45} C_VEL
LIN {X 0,Y 277.32,Z 813.638,A -85,B 0,C 180,E1 11122.651,E2 11122.651} C_VEL
LIN {X 0,Y 269.189,Z 829.465,A -85,B 0,C 180,E1 11119.587,E2 11119.587} C_VEL
LIN {X 0,Y 261.151,Z 844.431,A -85,B 0,C 180,E1 11116.033,E2 11116.033} C_VEL
LIN {X 0,Y 253.022,Z 859.658,A -85,B 0,C 180,E1 11111.593,E2 11111.593} C_VEL
LIN {X 0,Y 246.625,Z 872.107,A -85,B 0,C 180,E1 11107.158,E2 11107.158} C_VEL
LIN {X 0,Y 241.116,Z 883.669,A -85,B 0,C 180,E1 11102.055,E2 11102.055} C_VEL
LIN {X 0,Y 237.055,Z 893.653,A -85,B 0,C 180,E1 11096.596,E2 11096.596} C_VEL
LIN {X 0,Y 234.64,Z 901.549,A -85,B 0,C 180,E1 11091.233,E2 11091.233} C_VEL
LIN {X 0,Y 233.547,Z 907.28,A -85,B 0,C 180,E1 11086.155,E2 11086.155} C_VEL
LIN {X 0,Y 233.309,Z 911.433,A -85,B 0,C 180,E1 11081.367,E2 11081.367} C_VEL
LIN {X 0,Y 233.56,Z 914.246,A -85,B 0,C 180,E1 11076.388,E2 11076.388} C_VEL
LIN {X 0,Y 233.781,Z 915.395,A -85,B 0,C 180,E1 11072.449,E2 11072.449} C_VEL
LIN {X 0,Y 233.814,Z 915.554,A -85,B 0,C 180,E1 11068.772,E2 11068.772} C_VEL
LIN {X 0,Y 233.631,Z 914.735,A -85,B 0,C 180,E1 11064.841,E2 11064.841} C_VEL
LIN {X 0,Y 233.339,Z 912.485,A -85,B 0,C 180,E1 11060.128,E2 11060.128} C_VEL
LIN {X 0,Y 233.425,Z 908.71,A -85,B 0,C 180,E1 11055.359,E2 11055.359} C_VEL
LIN {X 0,Y 234.231,Z 903.321,A -85,B 0,C 180,E1 11050.29,E2 11050.29} C_VEL
LIN {X 0,Y 236.129,Z 896.185,A -85,B 0,C 180,E1 11045.213,E2 11045.213} C_VEL
LIN {X 0,Y 239.289,Z 887.474,A -85,B 0,C 180,E1 11040.18,E2 11040.18} C_VEL
LIN {X 0,Y 243.832,Z 876.785,A -85,B 0,C 180,E1 11035.248,E2 11035.248} C_VEL
LIN {X 0,Y 249.802,Z 864.031,A -85,B 0,C 180,E1 11030.472,E2 11030.472} C_VEL
LIN {X 0,Y 256.43,Z 850.617,A -85,B 0,C 180,E1 11026.356,E2 11026.356} C_VEL
LIN {X 0,Y 263.936,Z 835.305,A -85,B 0,C 180,E1 11022.537,E2 11022.537} C_VEL
LIN {X 0,Y 271.692,Z 818.993,A -85,B 0,C 180,E1 11019.223,E2 11019.223} C_VEL
LIN {X 0,Y 279.442,Z 801.995,A -85,B 0,C 180,E1 11016.381,E2 11016.381} C_VEL
LIN {X 0,Y 286.909,Z 784.21,A -85,B 0,C 180,E1 11013.959,E2 11013.959} C_VEL
LIN {X 0,Y 294.219,Z 765.111,A -85,B 0,C 180,E1 11011.831,E2 11011.831} C_VEL
LIN {X 0,Y 300.936,Z 745.482,A -85,B 0,C 180,E1 11010.056,E2 11010.056} C_VEL
LIN {X 0,Y 306.904,Z 725.034,A -85,B 0,C 180,E1 11008.595,E2 11008.595} C_VEL
LIN {X 0,Y 312.256,Z 703.193,A -85,B 0,C 180,E1 11007.37,E2 11007.37} C_VEL
LIN {X 0,Y 316.489,Z 681.898,A -85,B 0,C 180,E1 11006.464,E2 11006.464} C_VEL
LIN {X 0,Y 319.59,Z 659.537,A -85,B 0,C 180,E1 11005.776,E2 11005.776} C_VEL
LIN {X 0,Y 321.879,Z 628.927,A -85,B 0,C 180,E1 11005.088,E2 11005.088} C_VEL
LIN {X 0,Y 333.975,Z 442.714,A -85,B 0,C 180,E1 11001.244,E2 11001.244} C_VEL
LIN {X 0,Y 336.146,Z 410.51,A -85,B 0,C 180,E1 11000.548,E2 11000.548} C_VEL
LIN {X 0,Y 327.695,Z 397.583,A -85,B 0,C 180,E1 10997.628,E2 10997.628} C_VEL
LIN {X 0,Y 318.018,Z 383.694,A -85,B 0,C 180,E1 10993.871,E2 10993.871} C_VEL
LIN {X 0,Y 309.837,Z 372.933,A -85,B 0,C 180,E1 10990.224,E2 10990.224} C_VEL
LIN {X 0,Y 302.636,Z 363.9,A -85,B 0,C 180,E1 10986.546,E2 10986.546} C_VEL
LIN {X 0,Y 297.845,Z 358.285,A -85,B 0,C 180,E1 10983.754,E2 10983.754} C_VEL
LIN {X 0,Y 294.236,Z 354.021,A -85,B 0,C 180,E1 10981.364,E2 10981.364} C_VEL
LIN {X 0,Y 291.995,Z 350.971,A -85,B 0,C 180,E1 10979.187,E2 10979.187} C_VEL
LIN {X 0,Y 291.102,Z 349.164,A -85,B 0,C 180,E1 10977.835,E2 10977.835} C_VEL
LIN {X 0,Y 288.277,Z 344.155,A -85,B 0,C 180,E1 10972.741,E2 10972.741} C_VEL
LIN {X 0,Y 285.563,Z 339.921,A -85,B 0,C 180,E1 10964.152,E2 10964.152} C_VEL
LIN {X 0,Y 285.331,Z 339.361,A -85,B 0,C 180,E1 10959.91,E2 10959.91} C_VEL
LIN {X 0,Y 285.472,Z 340.396,A -85,B 0,C 180,E1 10956.029,E2 10956.029} C_VEL
LIN {X 0,Y 287.783,Z 344.326,A -85,B 0,C 180,E1 10948.347,E2 10948.347} C_VEL
LIN {X 0,Y 290.313,Z 349.315,A -85,B 0,C 180,E1 10943.369,E2 10943.369} C_VEL
LIN {X 0,Y 292.873,Z 354.41,A -85,B 0,C 180,E1 10939.561,E2 10939.561} C_VEL
LIN {X 0,Y 295.231,Z 359.197,A -85,B 0,C 180,E1 10936.569,E2 10936.569} C_VEL
LIN {X 0,Y 297.821,Z 364.436,A -85,B 0,C 180,E1 10933.758,E2 10933.758} C_VEL
LIN {X 0,Y 300.959,Z 371.093,A -85,B 0,C 180,E1 10930.631,E2 10930.631} C_VEL
LIN {X 0,Y 305.394,Z 380.717,A -85,B 0,C 180,E1 10926.895,E2 10926.895} C_VEL
LIN {X 0,Y 312.226,Z 392.327,A -85,B 0,C 180,E1 10923.593,E2 10923.593} C_VEL
LIN {X 0,Y 318.219,Z 403.237,A -85,B 0,C 180,E1 10920.983,E2 10920.983} C_VEL
LIN {X 0,Y 319.38,Z 469.999,A -85,B 0,C 180,E1 10917.487,E2 10917.487} C_VEL
LIN {X 0,Y 305.487,Z 635.457,A -85,B 0,C 180,E1 10913.71,E2 10913.71} C_VEL
LIN {X 0,Y 302.661,Z 656.972,A -85,B 0,C 180,E1 10912.997,E2 10912.997} C_VEL
LIN {X 0,Y 298.897,Z 677.631,A -85,B 0,C 180,E1 10912.005,E2 10912.005} C_VEL
LIN {X 0,Y 294.225,Z 697.817,A -85,B 0,C 180,E1 10910.699,E2 10910.699} C_VEL
LIN {X 0,Y 288.841,Z 717.015,A -85,B 0,C 180,E1 10909.091,E2 10909.091} C_VEL
LIN {X 0,Y 282.633,Z 735.918,A -85,B 0,C 180,E1 10907.077,E2 10907.077} C_VEL
LIN {X 0,Y 275.967,Z 753.727,A -85,B 0,C 180,E1 10904.682,E2 10904.682} C_VEL
LIN {X 0,Y 269.354,Z 769.647,A -85,B 0,C 180,E1 10902,E2 10902} C_VEL
LIN {X 0,Y 262.838,Z 784.094,A -85,B 0,C 180,E1 10898.975,E2 10898.975} C_VEL
LIN {X 0,Y 256.598,Z 797.095,A -85,B 0,C 180,E1 10895.593,E2 10895.593} C_VEL
LIN {X 0,Y 251.116,Z 808.12,A -85,B 0,C 180,E1 10892.027,E2 10892.027} C_VEL
LIN {X 0,Y 246.109,Z 818.053,A -85,B 0,C 180,E1 10887.998,E2 10887.998} C_VEL
LIN {X 0,Y 241.892,Z 826.515,A -85,B 0,C 180,E1 10883.595,E2 10883.595} C_VEL
LIN {X 0,Y 238.695,Z 833.319,A -85,B 0,C 180,E1 10878.893,E2 10878.893} C_VEL
LIN {X 0,Y 236.583,Z 838.309,A -85,B 0,C 180,E1 10874.058,E2 10874.058} C_VEL
LIN {X 0,Y 235.451,Z 841.586,A -85,B 0,C 180,E1 10869.102,E2 10869.102} C_VEL
LIN {X 0,Y 235.152,Z 843.133,A -85,B 0,C 180,E1 10864.301,E2 10864.301} C_VEL
LIN {X 0,Y 235.579,Z 843.14,A -85,B 0,C 180,E1 10859.385,E2 10859.385} C_VEL
LIN {X 0,Y 236.882,Z 841.484,A -85,B 0,C 180,E1 10854.378,E2 10854.378} C_VEL
LIN {X 0,Y 239.215,Z 838.179,A -85,B 0,C 180,E1 10849.525,E2 10849.525} C_VEL
LIN {X 0,Y 242.701,Z 833.162,A -85,B 0,C 180,E1 10844.785,E2 10844.785} C_VEL
LIN {X 0,Y 247.449,Z 826.335,A -85,B 0,C 180,E1 10840.214,E2 10840.214} C_VEL
LIN {X 0,Y 253.226,Z 817.859,A -85,B 0,C 180,E1 10835.964,E2 10835.964} C_VEL
LIN {X 0,Y 260.221,Z 807.232,A -85,B 0,C 180,E1 10831.885,E2 10831.885} C_VEL
LIN {X 0,Y 267.849,Z 794.996,A -85,B 0,C 180,E1 10828.247,E2 10828.247} C_VEL
LIN {X 0,Y 275.576,Z 781.694,A -85,B 0,C 180,E1 10825.118,E2 10825.118} C_VEL
LIN {X 0,Y 283.324,Z 767.197,A -85,B 0,C 180,E1 10822.398,E2 10822.398} C_VEL
LIN {X 0,Y 291.02,Z 751.354,A -85,B 0,C 180,E1 10820.012,E2 10820.012} C_VEL
LIN {X 0,Y 298.466,Z 734.167,A -85,B 0,C 180,E1 10817.945,E2 10817.945} C_VEL
LIN {X 0,Y 300.257,Z 729.754,A -85,B 0,C 180,E1 10817.481,E2 10817.481} C_VEL
LIN {X 0,Y 302.249,Z 723.501,A -85,B 0,C 180,E1 10816.69,E2 10816.69} C_VEL
LIN {X 0,Y 305.037,Z 707.921,A -85,B 0,C 180,E1 10814.354,E2 10814.354} C_VEL
LIN {X 0,Y 306.731,Z 701.249,A -85,B 0,C 180,E1 10813.695,E2 10813.695} C_VEL
LIN {X 0,Y 312.099,Z 682.157,A -85,B 0,C 180,E1 10812.542,E2 10812.542} C_VEL
LIN {X 0,Y 316.78,Z 661.17,A -85,B 0,C 180,E1 10811.593,E2 10811.593} C_VEL
LIN {X 0,Y 320.237,Z 639.625,A -85,B 0,C 180,E1 10810.917,E2 10810.917} C_VEL
LIN {X 0,Y 337.491,Z 475.01,A -85,B 0,C 180,E1 10807.275,E2 10807.275} C_VEL
LIN {X 0,Y 339.789,Z 424.646,A -85,B 0,C 180,E1 10804.419,E2 10804.419} C_VEL
LIN {X 0,Y 337.044,Z 416.68,A -85,B 0,C 180,E1 10801.437,E2 10801.437} C_VEL
LIN {X 0,Y 335.413,Z 411.501,A -85,B 0,C 180,E1 10798.718,E2 10798.718} C_VEL
LIN {X 0,Y 334.691,Z 408.536,A -85,B 0,C 180,E1 10796.403,E2 10796.403} C_VEL
LIN {X 0,Y 334.821,Z 405.836,A -85,B 0,C 180,E1 10792.794,E2 10792.794} C_VEL
LIN {X 0,Y 336.04,Z 406.391,A -85,B 0,C 180,E1 10789.716,E2 10789.716} C_VEL
LIN {X 0,Y 339.045,Z 410.717,A -85,B 0,C 180,E1 10785.918,E2 10785.918} C_VEL
LIN {X 0,Y 341.525,Z 414.729,A -85,B 0,C 180,E1 10783.773,E2 10783.773} C_VEL
LIN {X 0,Y 344.688,Z 420.169,A -85,B 0,C 180,E1 10781.567,E2 10781.567} C_VEL
LIN {X 0,Y 344.73,Z 420.962,A -85,B 0,C 180,E1 10781.491,E2 10781.491} C_VEL
LIN {X 0,Y 331.152,Z 580.309,A -85,B 0,C 180,E1 10778.173,E2 10778.173} C_VEL
LIN {X 0,Y 325.299,Z 653.595,A -85,B 0,C 180,E1 10776.632,E2 10776.632} C_VEL
LIN {X 0,Y 321.927,Z 675.914,A -85,B 0,C 180,E1 10775.997,E2 10775.997} C_VEL
LIN {X 0,Y 317.271,Z 697.542,A -85,B 0,C 180,E1 10775.172,E2 10775.172} C_VEL
LIN {X 0,Y 311.558,Z 718.716,A -85,B 0,C 180,E1 10774.082,E2 10774.082} C_VEL
LIN {X 0,Y 304.867,Z 739.223,A -85,B 0,C 180,E1 10772.716,E2 10772.716} C_VEL
LIN {X 0,Y 297.52,Z 758.513,A -85,B 0,C 180,E1 10771.092,E2 10771.092} C_VEL
LIN {X 0,Y 289.484,Z 777.375,A -85,B 0,C 180,E1 10769.121,E2 10769.121} C_VEL
LIN {X 0,Y 280.584,Z 796.183,A -85,B 0,C 180,E1 10766.678,E2 10766.678} C_VEL
LIN {X 0,Y 271.904,Z 813.034,A -85,B 0,C 180,E1 10763.959,E2 10763.959} C_VEL
LIN {X 0,Y 263.212,Z 829.151,A -85,B 0,C 180,E1 10760.794,E2 10760.794} C_VEL
LIN {X 0,Y 254.828,Z 844.009,A -85,B 0,C 180,E1 10757.195,E2 10757.195} C_VEL
LIN {X 0,Y 246.682,Z 858.404,A -85,B 0,C 180,E1 10752.913,E2 10752.913} C_VEL
LIN {X 0,Y 239.551,Z 871.419,A -85,B 0,C 180,E1 10748.147,E2 10748.147} C_VEL
LIN {X 0,Y 233.87,Z 882.581,A -85,B 0,C 180,E1 10743.075,E2 10743.075} C_VEL
LIN {X 0,Y 229.52,Z 892.456,A -85,B 0,C 180,E1 10737.498,E2 10737.498} C_VEL
LIN {X 0,Y 226.884,Z 900.291,A -85,B 0,C 180,E1 10731.996,E2 10731.996} C_VEL
LIN {X 0,Y 225.654,Z 906.036,A -85,B 0,C 180,E1 10726.736,E2 10726.736} C_VEL
LIN {X 0,Y 225.362,Z 910.403,A -85,B 0,C 180,E1 10721.514,E2 10721.514} C_VEL
LIN {X 0,Y 225.64,Z 913.116,A -85,B 0,C 180,E1 10716.358,E2 10716.358} C_VEL
LIN {X 0,Y 225.878,Z 914.212,A -85,B 0,C 180,E1 10712.281,E2 10712.281} C_VEL
LIN {X 0,Y 225.894,Z 914.287,A -85,B 0,C 180,E1 10708.222,E2 10708.222} C_VEL
LIN {X 0,Y 225.632,Z 913.173,A -85,B 0,C 180,E1 10703.637,E2 10703.637} C_VEL
LIN {X 0,Y 225.382,Z 910.391,A -85,B 0,C 180,E1 10698.645,E2 10698.645} C_VEL
LIN {X 0,Y 225.608,Z 906.413,A -85,B 0,C 180,E1 10693.785,E2 10693.785} C_VEL
LIN {X 0,Y 226.842,Z 900.228,A -85,B 0,C 180,E1 10688.266,E2 10688.266} C_VEL
LIN {X 0,Y 229.247,Z 892.729,A -85,B 0,C 180,E1 10683.023,E2 10683.023} C_VEL
LIN {X 0,Y 233.046,Z 883.343,A -85,B 0,C 180,E1 10677.856,E2 10677.856} C_VEL
LIN {X 0,Y 238.308,Z 872.116,A -85,B 0,C 180,E1 10672.828,E2 10672.828} C_VEL
LIN {X 0,Y 244.336,Z 860.159,A -85,B 0,C 180,E1 10668.474,E2 10668.474} C_VEL
LIN {X 0,Y 251.535,Z 846.127,A -85,B 0,C 180,E1 10664.313,E2 10664.313} C_VEL
LIN {X 0,Y 259.401,Z 830.767,A -85,B 0,C 180,E1 10660.592,E2 10660.592} C_VEL
LIN {X 0,Y 267.14,Z 815.034,A -85,B 0,C 180,E1 10657.486,E2 10657.486} C_VEL
LIN {X 0,Y 275.276,Z 797.414,A -85,B 0,C 180,E1 10654.642,E2 10654.642} C_VEL
LIN {X 0,Y 283.136,Z 779.012,A -85,B 0,C 180,E1 10652.225,E2 10652.225} C_VEL
LIN {X 0,Y 290.406,Z 760.002,A -85,B 0,C 180,E1 10650.207,E2 10650.207} C_VEL
LIN {X 0,Y 297.046,Z 740.409,A -85,B 0,C 180,E1 10648.532,E2 10648.532} C_VEL
LIN {X 0,Y 302.992,Z 720.252,A -85,B 0,C 180,E1 10647.144,E2 10647.144} C_VEL
LIN {X 0,Y 308.165,Z 698.691,A -85,B 0,C 180,E1 10646.004,E2 10646.004} C_VEL
LIN {X 0,Y 312.448,Z 676.088,A -85,B 0,C 180,E1 10645.117,E2 10645.117} C_VEL
LIN {X 0,Y 315.339,Z 653.984,A -85,B 0,C 180,E1 10644.478,E2 10644.478} C_VEL
LIN {X 0,Y 329.141,Z 449.605,A -85,B 0,C 180,E1 10640.224,E2 10640.224} C_VEL
LIN {X 0,Y 331.556,Z 414.709,A -85,B 0,C 180,E1 10639.465,E2 10639.465} C_VEL
LIN {X 0,Y 322.903,Z 401.387,A -85,B 0,C 180,E1 10636.321,E2 10636.321} C_VEL
LIN {X 0,Y 314.587,Z 389.548,A -85,B 0,C 180,E1 10632.949,E2 10632.949} C_VEL
LIN {X 0,Y 307.601,Z 380.142,A -85,B 0,C 180,E1 10629.732,E2 10629.732} C_VEL
LIN {X 0,Y 300.581,Z 371.153,A -85,B 0,C 180,E1 10626.025,E2 10626.025} C_VEL
LIN {X 0,Y 295.984,Z 365.698,A -85,B 0,C 180,E1 10623.293,E2 10623.293} C_VEL
LIN {X 0,Y 292.47,Z 361.48,A -85,B 0,C 180,E1 10620.882,E2 10620.882} C_VEL
LIN {X 0,Y 288.219,Z 356.545,A -85,B 0,C 180,E1 10617.597,E2 10617.597} C_VEL
LIN {X 0,Y 285.874,Z 353.832,A -85,B 0,C 180,E1 10614.985,E2 10614.985} C_VEL
LIN {X 0,Y 284.789,Z 351.324,A -85,B 0,C 180,E1 10612.537,E2 10612.537} C_VEL
LIN {X 0,Y 282.247,Z 347.271,A -85,B 0,C 180,E1 10604.382,E2 10604.382} C_VEL
LIN {X 0,Y 282.001,Z 346.613,A -85,B 0,C 180,E1 10600.533,E2 10600.533} C_VEL
LIN {X 0,Y 282.091,Z 347.432,A -85,B 0,C 180,E1 10596.612,E2 10596.612} C_VEL
LIN {X 0,Y 284.248,Z 351.363,A -85,B 0,C 180,E1 10588.629,E2 10588.629} C_VEL
LIN {X 0,Y 286.666,Z 356.316,A -85,B 0,C 180,E1 10583.635,E2 10583.635} C_VEL
LIN {X 0,Y 289.095,Z 361.311,A -85,B 0,C 180,E1 10579.851,E2 10579.851} C_VEL
LIN {X 0,Y 291.495,Z 366.355,A -85,B 0,C 180,E1 10576.686,E2 10576.686} C_VEL
LIN {X 0,Y 294.016,Z 371.571,A -85,B 0,C 180,E1 10573.869,E2 10573.869} C_VEL
LIN {X 0,Y 297.263,Z 378.411,A -85,B 0,C 180,E1 10570.735,E2 10570.735} C_VEL
LIN {X 0,Y 303.876,Z 389.261,A -85,B 0,C 180,E1 10567,E2 10567} C_VEL
LIN {X 0,Y 309.893,Z 399.784,A -85,B 0,C 180,E1 10564.027,E2 10564.027} C_VEL
LIN {X 0,Y 314.308,Z 408.116,A -85,B 0,C 180,E1 10562.031,E2 10562.031} C_VEL
LIN {X 0,Y 315.035,Z 471.395,A -85,B 0,C 180,E1 10558.686,E2 10558.686} C_VEL
LIN {X 0,Y 300.758,Z 636.205,A -85,B 0,C 180,E1 10554.923,E2 10554.923} C_VEL
LIN {X 0,Y 297.85,Z 657.574,A -85,B 0,C 180,E1 10554.211,E2 10554.211} C_VEL
LIN {X 0,Y 294.029,Z 677.928,A -85,B 0,C 180,E1 10553.234,E2 10553.234} C_VEL
LIN {X 0,Y 289.207,Z 698.174,A -85,B 0,C 180,E1 10551.926,E2 10551.926} C_VEL
LIN {X 0,Y 283.538,Z 717.76,A -85,B 0,C 180,E1 10550.283,E2 10550.283} C_VEL
LIN {X 0,Y 277.212,Z 736.394,A -85,B 0,C 180,E1 10548.29,E2 10548.29} C_VEL
LIN {X 0,Y 270.317,Z 754.197,A -85,B 0,C 180,E1 10545.887,E2 10545.887} C_VEL
LIN {X 0,Y 263.407,Z 770.249,A -85,B 0,C 180,E1 10543.167,E2 10543.167} C_VEL
LIN {X 0,Y 256.603,Z 784.761,A -85,B 0,C 180,E1 10540.101,E2 10540.101} C_VEL
LIN {X 0,Y 250.066,Z 797.826,A -85,B 0,C 180,E1 10536.661,E2 10536.661} C_VEL
LIN {X 0,Y 244.3,Z 808.91,A -85,B 0,C 180,E1 10533.025,E2 10533.025} C_VEL
LIN {X 0,Y 238.9,Z 819.105,A -85,B 0,C 180,E1 10528.803,E2 10528.803} C_VEL
LIN {X 0,Y 234.524,Z 827.432,A -85,B 0,C 180,E1 10524.375,E2 10524.375} C_VEL
LIN {X 0,Y 231.102,Z 834.289,A -85,B 0,C 180,E1 10519.533,E2 10519.533} C_VEL
LIN {X 0,Y 228.824,Z 839.34,A -85,B 0,C 180,E1 10514.544,E2 10514.544} C_VEL
LIN {X 0,Y 227.622,Z 842.544,A -85,B 0,C 180,E1 10509.698,E2 10509.698} C_VEL
LIN {X 0,Y 227.242,Z 844.269,A -85,B 0,C 180,E1 10504.739,E2 10504.739} C_VEL
LIN {X 0,Y 227.636,Z 844.473,A -85,B 0,C 180,E1 10499.664,E2 10499.664} C_VEL
LIN {X 0,Y 228.837,Z 843.179,A -85,B 0,C 180,E1 10494.782,E2 10494.782} C_VEL
LIN {X 0,Y 231.262,Z 840.052,A -85,B 0,C 180,E1 10489.574,E2 10489.574} C_VEL
LIN {X 0,Y 235.064,Z 834.964,A -85,B 0,C 180,E1 10484.394,E2 10484.394} C_VEL
LIN {X 0,Y 240.153,Z 828.124,A -85,B 0,C 180,E1 10479.567,E2 10479.567} C_VEL
LIN {X 0,Y 246.53,Z 819.323,A -85,B 0,C 180,E1 10474.995,E2 10474.995} C_VEL
LIN {X 0,Y 254.006,Z 808.597,A -85,B 0,C 180,E1 10470.778,E2 10470.778} C_VEL
LIN {X 0,Y 261.832,Z 796.706,A -85,B 0,C 180,E1 10467.163,E2 10467.163} C_VEL
LIN {X 0,Y 269.707,Z 783.819,A -85,B 0,C 180,E1 10464.065,E2 10464.065} C_VEL
LIN {X 0,Y 277.895,Z 769.331,A -85,B 0,C 180,E1 10461.279,E2 10461.279} C_VEL
LIN {X 0,Y 286.2,Z 753.049,A -85,B 0,C 180,E1 10458.79,E2 10458.79} C_VEL
LIN {X 0,Y 294.264,Z 735.222,A -85,B 0,C 180,E1 10456.636,E2 10456.636} C_VEL
LIN {X 0,Y 301.152,Z 717.756,A -85,B 0,C 180,E1 10454.96,E2 10454.96} C_VEL
LIN {X 0,Y 306.731,Z 701.249,A -85,B 0,C 180,E1 10453.695,E2 10453.695} C_VEL
LIN {X 0,Y 308.44,Z 694.451,A -85,B 0,C 180,E1 10453.07,E2 10453.07} C_VEL
LIN {X 0,Y 310.684,Z 677.549,A -85,B 0,C 180,E1 10451.102,E2 10451.102} C_VEL
LIN {X 0,Y 311.938,Z 670.43,A -85,B 0,C 180,E1 10450.6,E2 10450.6} C_VEL
LIN {X 0,Y 315.902,Z 649.75,A -85,B 0,C 180,E1 10449.848,E2 10449.848} C_VEL
LIN {X 0,Y 319.375,Z 622.142,A -85,B 0,C 180,E1 10449.165,E2 10449.165} C_VEL
LIN {X 0,Y 334.977,Z 476.197,A -85,B 0,C 180,E1 10445.985,E2 10445.985} C_VEL
LIN {X 0,Y 337.49,Z 430.325,A -85,B 0,C 180,E1 10443.375,E2 10443.375} C_VEL
LIN {X 0,Y 335.376,Z 423.447,A -85,B 0,C 180,E1 10440.683,E2 10440.683} C_VEL
LIN {X 0,Y 334.031,Z 418.699,A -85,B 0,C 180,E1 10438.027,E2 10438.027} C_VEL
LIN {X 0,Y 333.556,Z 416.251,A -85,B 0,C 180,E1 10436.046,E2 10436.046} C_VEL
LIN {X 0,Y 333.818,Z 413.763,A -85,B 0,C 180,E1 10432.6,E2 10432.6} C_VEL
LIN {X 0,Y 334.918,Z 414.302,A -85,B 0,C 180,E1 10429.855,E2 10429.855} C_VEL
LIN {X 0,Y 337.707,Z 418.459,A -85,B 0,C 180,E1 10426.186,E2 10426.186} C_VEL
LIN {X 0,Y 340.088,Z 422.475,A -85,B 0,C 180,E1 10424.044,E2 10424.044} C_VEL
LIN {X 0,Y 341.895,Z 425.858,A -85,B 0,C 180,E1 10422.67,E2 10422.67} C_VEL
LIN {X 0,Y 328.111,Z 580.339,A -85,B 0,C 180,E1 10419.463,E2 10419.463} C_VEL
LIN {X 0,Y 322.011,Z 653.266,A -85,B 0,C 180,E1 10417.933,E2 10417.933} C_VEL
LIN {X 0,Y 318.531,Z 675.485,A -85,B 0,C 180,E1 10417.305,E2 10417.305} C_VEL
LIN {X 0,Y 313.733,Z 697.04,A -85,B 0,C 180,E1 10416.493,E2 10416.493} C_VEL
LIN {X 0,Y 307.846,Z 718.198,A -85,B 0,C 180,E1 10415.419,E2 10415.419} C_VEL
LIN {X 0,Y 301.168,Z 738.066,A -85,B 0,C 180,E1 10414.113,E2 10414.113} C_VEL
LIN {X 0,Y 293.643,Z 757.217,A -85,B 0,C 180,E1 10412.524,E2 10412.524} C_VEL
LIN {X 0,Y 285.278,Z 776.244,A -85,B 0,C 180,E1 10410.565,E2 10410.565} C_VEL
LIN {X 0,Y 276.36,Z 794.353,A -85,B 0,C 180,E1 10408.231,E2 10408.231} C_VEL
LIN {X 0,Y 267.059,Z 811.756,A -85,B 0,C 180,E1 10405.449,E2 10405.449} C_VEL
LIN {X 0,Y 257.703,Z 828.262,A -85,B 0,C 180,E1 10402.191,E2 10402.191} C_VEL
LIN {X 0,Y 248.619,Z 843.637,A -85,B 0,C 180,E1 10398.415,E2 10398.415} C_VEL
LIN {X 0,Y 240.065,Z 857.865,A -85,B 0,C 180,E1 10394.067,E2 10394.067} C_VEL
LIN {X 0,Y 232.553,Z 870.756,A -85,B 0,C 180,E1 10389.196,E2 10389.196} C_VEL
LIN {X 0,Y 226.359,Z 882.198,A -85,B 0,C 180,E1 10383.815,E2 10383.815} C_VEL
LIN {X 0,Y 221.888,Z 891.615,A -85,B 0,C 180,E1 10378.235,E2 10378.235} C_VEL
LIN {X 0,Y 218.964,Z 899.654,A -85,B 0,C 180,E1 10372.269,E2 10372.269} C_VEL
LIN {X 0,Y 217.732,Z 905.049,A -85,B 0,C 180,E1 10367.088,E2 10367.088} C_VEL
LIN {X 0,Y 217.421,Z 909.489,A -85,B 0,C 180,E1 10361.402,E2 10361.402} C_VEL
LIN {X 0,Y 217.697,Z 911.889,A -85,B 0,C 180,E1 10356.591,E2 10356.591} C_VEL
LIN {X 0,Y 217.965,Z 912.987,A -85,B 0,C 180,E1 10352.363,E2 10352.363} C_VEL
LIN {X 0,Y 217.986,Z 913.054,A -85,B 0,C 180,E1 10348.157,E2 10348.157} C_VEL
LIN {X 0,Y 217.697,Z 911.902,A -85,B 0,C 180,E1 10343.404,E2 10343.404} C_VEL
LIN {X 0,Y 217.446,Z 909.144,A -85,B 0,C 180,E1 10338.325,E2 10338.325} C_VEL
LIN {X 0,Y 217.691,Z 905.3,A -85,B 0,C 180,E1 10333.452,E2 10333.452} C_VEL
LIN {X 0,Y 219.019,Z 899.14,A -85,B 0,C 180,E1 10327.731,E2 10327.731} C_VEL
LIN {X 0,Y 221.72,Z 891.348,A -85,B 0,C 180,E1 10322.114,E2 10322.114} C_VEL
LIN {X 0,Y 225.893,Z 881.741,A -85,B 0,C 180,E1 10316.709,E2 10316.709} C_VEL
LIN {X 0,Y 231.871,Z 869.761,A -85,B 0,C 180,E1 10311.296,E2 10311.296} C_VEL
LIN {X 0,Y 238.36,Z 857.624,A -85,B 0,C 180,E1 10306.86,E2 10306.86} C_VEL
LIN {X 0,Y 246.05,Z 843.276,A -85,B 0,C 180,E1 10302.646,E2 10302.646} C_VEL
LIN {X 0,Y 254.39,Z 827.558,A -85,B 0,C 180,E1 10298.899,E2 10298.899} C_VEL
LIN {X 0,Y 262.537,Z 811.529,A -85,B 0,C 180,E1 10295.784,E2 10295.784} C_VEL
LIN {X 0,Y 270.764,Z 794.027,A -85,B 0,C 180,E1 10293.041,E2 10293.041} C_VEL
LIN {X 0,Y 278.921,Z 775.181,A -85,B 0,C 180,E1 10290.643,E2 10290.643} C_VEL
LIN {X 0,Y 286.477,Z 755.823,A -85,B 0,C 180,E1 10288.646,E2 10288.646} C_VEL
LIN {X 0,Y 293.047,Z 736.399,A -85,B 0,C 180,E1 10287.059,E2 10287.059} C_VEL
LIN {X 0,Y 299.247,Z 714.926,A -85,B 0,C 180,E1 10285.667,E2 10285.667} C_VEL
LIN {X 0,Y 304.375,Z 693.313,A -85,B 0,C 180,E1 10284.586,E2 10284.586} C_VEL
LIN {X 0,Y 308.332,Z 671.506,A -85,B 0,C 180,E1 10283.794,E2 10283.794} C_VEL
LIN {X 0,Y 310.986,Z 648.951,A -85,B 0,C 180,E1 10283.184,E2 10283.184} C_VEL
LIN {X 0,Y 324.924,Z 449.306,A -85,B 0,C 180,E1 10279.026,E2 10279.026} C_VEL
LIN {X 0,Y 327.158,Z 419.115,A -85,B 0,C 180,E1 10278.395,E2 10278.395} C_VEL
LIN {X 0,Y 318.514,Z 405.731,A -85,B 0,C 180,E1 10275.103,E2 10275.103} C_VEL
LIN {X 0,Y 309.744,Z 393.1,A -85,B 0,C 180,E1 10271.31,E2 10271.31} C_VEL
LIN {X 0,Y 302.243,Z 383.229,A -85,B 0,C 180,E1 10267.605,E2 10267.605} C_VEL
LIN {X 0,Y 296.9,Z 376.427,A -85,B 0,C 180,E1 10264.55,E2 10264.55} C_VEL
LIN {X 0,Y 290.981,Z 369.197,A -85,B 0,C 180,E1 10260.589,E2 10260.589} C_VEL
LIN {X 0,Y 286.669,Z 364.186,A -85,B 0,C 180,E1 10257.202,E2 10257.202} C_VEL
LIN {X 0,Y 282.34,Z 359.186,A -85,B 0,C 180,E1 10252.881,E2 10252.881} C_VEL
LIN {X 0,Y 279.818,Z 356.776,A -85,B 0,C 180,E1 10248.876,E2 10248.876} C_VEL
LIN {X 0,Y 278.83,Z 354.184,A -85,B 0,C 180,E1 10243.116,E2 10243.116} C_VEL
LIN {X 0,Y 278.619,Z 353.997,A -85,B 0,C 180,E1 10239.191,E2 10239.191} C_VEL
LIN {X 0,Y 278.801,Z 355.397,A -85,B 0,C 180,E1 10235.142,E2 10235.142} C_VEL
LIN {X 0,Y 280.757,Z 358.61,A -85,B 0,C 180,E1 10228.731,E2 10228.731} C_VEL
LIN {X 0,Y 283.048,Z 363.399,A -85,B 0,C 180,E1 10223.85,E2 10223.85} C_VEL
LIN {X 0,Y 285.332,Z 368.26,A -85,B 0,C 180,E1 10220.115,E2 10220.115} C_VEL
LIN {X 0,Y 287.58,Z 373.092,A -85,B 0,C 180,E1 10217.044,E2 10217.044} C_VEL
LIN {X 0,Y 289.994,Z 377.385,A -85,B 0,C 180,E1 10214.816,E2 10214.816} C_VEL
LIN {X 0,Y 295.45,Z 386.119,A -85,B 0,C 180,E1 10211.079,E2 10211.079} C_VEL
LIN {X 0,Y 301.609,Z 396.468,A -85,B 0,C 180,E1 10207.522,E2 10207.522} C_VEL
LIN {X 0,Y 307.305,Z 406.727,A -85,B 0,C 180,E1 10204.599,E2 10204.599} C_VEL
LIN {X 0,Y 310.47,Z 412.877,A -85,B 0,C 180,E1 10203.111,E2 10203.111} C_VEL
LIN {X 0,Y 310.81,Z 472.668,A -85,B 0,C 180,E1 10199.918,E2 10199.918} C_VEL
LIN {X 0,Y 296.208,Z 636.499,A -85,B 0,C 180,E1 10196.185,E2 10196.185} C_VEL
LIN {X 0,Y 293.196,Z 658.023,A -85,B 0,C 180,E1 10195.47,E2 10195.47} C_VEL
LIN {X 0,Y 289.299,Z 678.21,A -85,B 0,C 180,E1 10194.505,E2 10194.505} C_VEL
LIN {X 0,Y 284.326,Z 698.527,A -85,B 0,C 180,E1 10193.197,E2 10193.197} C_VEL
LIN {X 0,Y 278.361,Z 718.513,A -85,B 0,C 180,E1 10191.519,E2 10191.519} C_VEL
LIN {X 0,Y 271.92,Z 736.878,A -85,B 0,C 180,E1 10189.551,E2 10189.551} C_VEL
LIN {X 0,Y 264.766,Z 754.74,A -85,B 0,C 180,E1 10187.133,E2 10187.133} C_VEL
LIN {X 0,Y 257.327,Z 771.378,A -85,B 0,C 180,E1 10184.286,E2 10184.286} C_VEL
LIN {X 0,Y 250.022,Z 786.306,A -85,B 0,C 180,E1 10181.069,E2 10181.069} C_VEL
LIN {X 0,Y 243.005,Z 799.687,A -85,B 0,C 180,E1 10177.439,E2 10177.439} C_VEL
LIN {X 0,Y 236.558,Z 811.45,A -85,B 0,C 180,E1 10173.395,E2 10173.395} C_VEL
LIN {X 0,Y 230.989,Z 821.431,A -85,B 0,C 180,E1 10169.01,E2 10169.01} C_VEL
LIN {X 0,Y 226.53,Z 829.512,A -85,B 0,C 180,E1 10164.43,E2 10164.43} C_VEL
LIN {X 0,Y 223.222,Z 835.878,A -85,B 0,C 180,E1 10159.682,E2 10159.682} C_VEL
LIN {X 0,Y 220.89,Z 840.846,A -85,B 0,C 180,E1 10154.513,E2 10154.513} C_VEL
LIN {X 0,Y 219.648,Z 844.093,A -85,B 0,C 180,E1 10149.206,E2 10149.206} C_VEL
LIN {X 0,Y 219.345,Z 845.627,A -85,B 0,C 180,E1 10144.052,E2 10144.052} C_VEL
LIN {X 0,Y 219.823,Z 845.683,A -85,B 0,C 180,E1 10139.074,E2 10139.074} C_VEL
LIN {X 0,Y 221.198,Z 844.298,A -85,B 0,C 180,E1 10134.007,E2 10134.007} C_VEL
LIN {X 0,Y 223.706,Z 841.343,A -85,B 0,C 180,E1 10128.931,E2 10128.931} C_VEL
LIN {X 0,Y 227.779,Z 836.305,A -85,B 0,C 180,E1 10123.595,E2 10123.595} C_VEL
LIN {X 0,Y 233.123,Z 829.588,A -85,B 0,C 180,E1 10118.69,E2 10118.69} C_VEL
LIN {X 0,Y 239.91,Z 820.796,A -85,B 0,C 180,E1 10113.972,E2 10113.972} C_VEL
LIN {X 0,Y 247.087,Z 811.072,A -85,B 0,C 180,E1 10110.012,E2 10110.012} C_VEL
LIN {X 0,Y 255.036,Z 799.709,A -85,B 0,C 180,E1 10106.392,E2 10106.392} C_VEL
LIN {X 0,Y 263.581,Z 786.6,A -85,B 0,C 180,E1 10103.097,E2 10103.097} C_VEL
LIN {X 0,Y 272.359,Z 771.896,A -85,B 0,C 180,E1 10100.186,E2 10100.186} C_VEL
LIN {X 0,Y 280.425,Z 757.068,A -85,B 0,C 180,E1 10097.835,E2 10097.835} C_VEL
LIN {X 0,Y 288.73,Z 739.887,A -85,B 0,C 180,E1 10095.67,E2 10095.67} C_VEL
LIN {X 0,Y 296.529,Z 721.213,A -85,B 0,C 180,E1 10093.819,E2 10093.819} C_VEL
LIN {X 0,Y 303.117,Z 702.646,A -85,B 0,C 180,E1 10092.38,E2 10092.38} C_VEL
LIN {X 0,Y 308.87,Z 683.016,A -85,B 0,C 180,E1 10091.199,E2 10091.199} C_VEL
LIN {X 0,Y 311.938,Z 670.43,A -85,B 0,C 180,E1 10090.6,E2 10090.6} C_VEL
LIN {X 0,Y 313.179,Z 663.198,A -85,B 0,C 180,E1 10090.132,E2 10090.132} C_VEL
LIN {X 0,Y 314.384,Z 645.206,A -85,B 0,C 180,E1 10088.512,E2 10088.512} C_VEL
LIN {X 0,Y 315.036,Z 637.769,A -85,B 0,C 180,E1 10088.146,E2 10088.146} C_VEL
LIN {X 0,Y 332.713,Z 477.671,A -85,B 0,C 180,E1 10084.686,E2 10084.686} C_VEL
LIN {X 0,Y 335.377,Z 435.964,A -85,B 0,C 180,E1 10082.306,E2 10082.306} C_VEL
LIN {X 0,Y 333.594,Z 429.458,A -85,B 0,C 180,E1 10079.57,E2 10079.57} C_VEL
LIN {X 0,Y 332.636,Z 425.407,A -85,B 0,C 180,E1 10076.984,E2 10076.984} C_VEL
LIN {X 0,Y 332.413,Z 423.833,A -85,B 0,C 180,E1 10075.514,E2 10075.514} C_VEL
LIN {X 0,Y 332.822,Z 421.694,A -85,B 0,C 180,E1 10072.404,E2 10072.404} C_VEL
LIN {X 0,Y 333.798,Z 422.211,A -85,B 0,C 180,E1 10069.995,E2 10069.995} C_VEL
LIN {X 0,Y 336.332,Z 426.117,A -85,B 0,C 180,E1 10066.504,E2 10066.504} C_VEL
LIN {X 0,Y 338.653,Z 430.201,A -85,B 0,C 180,E1 10064.326,E2 10064.326} C_VEL
LIN {X 0,Y 339.208,Z 431.378,A -85,B 0,C 180,E1 10063.859,E2 10063.859} C_VEL
LIN {X 0,Y 324.545,Z 589.323,A -85,B 0,C 180,E1 10060.598,E2 10060.598} C_VEL
LIN {X 0,Y 318.917,Z 652.995,A -85,B 0,C 180,E1 10059.261,E2 10059.261} C_VEL
LIN {X 0,Y 315.269,Z 675.44,A -85,B 0,C 180,E1 10058.631,E2 10058.631} C_VEL
LIN {X 0,Y 310.415,Z 696.619,A -85,B 0,C 180,E1 10057.845,E2 10057.845} C_VEL
LIN {X 0,Y 304.528,Z 717.182,A -85,B 0,C 180,E1 10056.821,E2 10056.821} C_VEL
LIN {X 0,Y 297.906,Z 736.29,A -85,B 0,C 180,E1 10055.591,E2 10055.591} C_VEL
LIN {X 0,Y 289.856,Z 756.295,A -85,B 0,C 180,E1 10053.968,E2 10053.968} C_VEL
LIN {X 0,Y 281.618,Z 774.461,A -85,B 0,C 180,E1 10052.129,E2 10052.129} C_VEL
LIN {X 0,Y 272.025,Z 793.25,A -85,B 0,C 180,E1 10049.737,E2 10049.737} C_VEL
LIN {X 0,Y 262.352,Z 810.618,A -85,B 0,C 180,E1 10046.971,E2 10046.971} C_VEL
LIN {X 0,Y 252.775,Z 826.787,A -85,B 0,C 180,E1 10043.792,E2 10043.792} C_VEL
LIN {X 0,Y 243.546,Z 841.612,A -85,B 0,C 180,E1 10040.144,E2 10040.144} C_VEL
LIN {X 0,Y 234.437,Z 855.969,A -85,B 0,C 180,E1 10035.763,E2 10035.763} C_VEL
LIN {X 0,Y 226.656,Z 868.477,A -85,B 0,C 180,E1 10031.031,E2 10031.031} C_VEL
LIN {X 0,Y 219.889,Z 879.928,A -85,B 0,C 180,E1 10025.59,E2 10025.59} C_VEL
LIN {X 0,Y 214.859,Z 889.554,A -85,B 0,C 180,E1 10019.86,E2 10019.86} C_VEL
LIN {X 0,Y 211.585,Z 897.479,A -85,B 0,C 180,E1 10013.975,E2 10013.975} C_VEL
LIN {X 0,Y 209.904,Z 903.558,A -85,B 0,C 180,E1 10008.033,E2 10008.033} C_VEL
LIN {X 0,Y 209.471,Z 908.101,A -85,B 0,C 180,E1 10002.121,E2 10002.121} C_VEL
LIN {X 0,Y 209.752,Z 910.664,A -85,B 0,C 180,E1 9996.841,E2 9996.841} C_VEL
LIN {X 0,Y 210.051,Z 911.767,A -85,B 0,C 180,E1 9992.452,E2 9992.452} C_VEL
LIN {X 0,Y 210.08,Z 911.828,A -85,B 0,C 180,E1 9988.163,E2 9988.163} C_VEL
LIN {X 0,Y 209.78,Z 910.739,A -85,B 0,C 180,E1 9983.429,E2 9983.429} C_VEL
LIN {X 0,Y 209.51,Z 907.945,A -85,B 0,C 180,E1 9978.055,E2 9978.055} C_VEL
LIN {X 0,Y 209.82,Z 903.934,A -85,B 0,C 180,E1 9972.813,E2 9972.813} C_VEL
LIN {X 0,Y 211.321,Z 897.682,A -85,B 0,C 180,E1 9966.874,E2 9966.874} C_VEL
LIN {X 0,Y 214.165,Z 890.123,A -85,B 0,C 180,E1 9961.255,E2 9961.255} C_VEL
LIN {X 0,Y 218.564,Z 880.634,A -85,B 0,C 180,E1 9955.756,E2 9955.756} C_VEL
LIN {X 0,Y 224.904,Z 868.617,A -85,B 0,C 180,E1 9950.192,E2 9950.192} C_VEL
LIN {X 0,Y 231.737,Z 856.47,A -85,B 0,C 180,E1 9945.653,E2 9945.653} C_VEL
LIN {X 0,Y 239.328,Z 842.932,A -85,B 0,C 180,E1 9941.595,E2 9941.595} C_VEL
LIN {X 0,Y 248.241,Z 826.766,A -85,B 0,C 180,E1 9937.675,E2 9937.675} C_VEL
LIN {X 0,Y 256.697,Z 810.762,A -85,B 0,C 180,E1 9934.529,E2 9934.529} C_VEL
LIN {X 0,Y 265.213,Z 793.283,A -85,B 0,C 180,E1 9931.77,E2 9931.77} C_VEL
LIN {X 0,Y 273.688,Z 774.25,A -85,B 0,C 180,E1 9929.349,E2 9929.349} C_VEL
LIN {X 0,Y 281.453,Z 754.817,A -85,B 0,C 180,E1 9927.358,E2 9927.358} C_VEL
LIN {X 0,Y 288.22,Z 735.302,A -85,B 0,C 180,E1 9925.774,E2 9925.774} C_VEL
LIN {X 0,Y 294.526,Z 713.908,A -85,B 0,C 180,E1 9924.4,E2 9924.4} C_VEL
LIN {X 0,Y 299.714,Z 692.484,A -85,B 0,C 180,E1 9923.341,E2 9923.341} C_VEL
LIN {X 0,Y 303.743,Z 670.74,A -85,B 0,C 180,E1 9922.558,E2 9922.558} C_VEL
LIN {X 0,Y 306.423,Z 648.318,A -85,B 0,C 180,E1 9921.955,E2 9921.955} C_VEL
LIN {X 0,Y 320.752,Z 449.427,A -85,B 0,C 180,E1 9917.813,E2 9917.813} C_VEL
LIN {X 0,Y 322.721,Z 423.34,A -85,B 0,C 180,E1 9917.257,E2 9917.257} C_VEL
LIN {X 0,Y 314.206,Z 410.202,A -85,B 0,C 180,E1 9913.855,E2 9913.855} C_VEL
LIN {X 0,Y 306.925,Z 399.609,A -85,B 0,C 180,E1 9910.559,E2 9910.559} C_VEL
LIN {X 0,Y 300.039,Z 390.343,A -85,B 0,C 180,E1 9907.035,E2 9907.035} C_VEL
LIN {X 0,Y 293.945,Z 382.346,A -85,B 0,C 180,E1 9903.413,E2 9903.413} C_VEL
LIN {X 0,Y 288.966,Z 376.398,A -85,B 0,C 180,E1 9899.922,E2 9899.922} C_VEL
LIN {X 0,Y 284.998,Z 371.703,A -85,B 0,C 180,E1 9896.682,E2 9896.682} C_VEL
LIN {X 0,Y 280.507,Z 366.499,A -85,B 0,C 180,E1 9892.01,E2 9892.01} C_VEL
LIN {X 0,Y 275.607,Z 361.567,A -85,B 0,C 180,E1 9883.291,E2 9883.291} C_VEL
LIN {X 0,Y 275.272,Z 361.236,A -85,B 0,C 180,E1 9879.371,E2 9879.371} C_VEL
LIN {X 0,Y 275.408,Z 362.593,A -85,B 0,C 180,E1 9875.324,E2 9875.324} C_VEL
LIN {X 0,Y 277.244,Z 365.723,A -85,B 0,C 180,E1 9868.956,E2 9868.956} C_VEL
LIN {X 0,Y 279.53,Z 370.685,A -85,B 0,C 180,E1 9863.941,E2 9863.941} C_VEL
LIN {X 0,Y 282.535,Z 375.777,A -85,B 0,C 180,E1 9860.301,E2 9860.301} C_VEL
LIN {X 0,Y 286.438,Z 381.936,A -85,B 0,C 180,E1 9856.694,E2 9856.694} C_VEL
LIN {X 0,Y 292.28,Z 391.385,A -85,B 0,C 180,E1 9852.363,E2 9852.363} C_VEL
LIN {X 0,Y 298.859,Z 402.766,A -85,B 0,C 180,E1 9848.324,E2 9848.324} C_VEL
LIN {X 0,Y 304.578,Z 413.352,A -85,B 0,C 180,E1 9845.265,E2 9845.265} C_VEL
LIN {X 0,Y 306.702,Z 417.504,A -85,B 0,C 180,E1 9844.221,E2 9844.221} C_VEL
LIN {X 0,Y 306.714,Z 473.922,A -85,B 0,C 180,E1 9841.181,E2 9841.181} C_VEL
LIN {X 0,Y 291.733,Z 637.14,A -85,B 0,C 180,E1 9837.473,E2 9837.473} C_VEL
LIN {X 0,Y 288.636,Z 658.574,A -85,B 0,C 180,E1 9836.76,E2 9836.76} C_VEL
LIN {X 0,Y 284.544,Z 679.103,A -85,B 0,C 180,E1 9835.777,E2 9835.777} C_VEL
LIN {X 0,Y 279.579,Z 698.784,A -85,B 0,C 180,E1 9834.512,E2 9834.512} C_VEL
LIN {X 0,Y 273.656,Z 718.143,A -85,B 0,C 180,E1 9832.902,E2 9832.902} C_VEL
LIN {X 0,Y 267.05,Z 736.54,A -85,B 0,C 180,E1 9830.953,E2 9830.953} C_VEL
LIN {X 0,Y 260.304,Z 753.067,A -85,B 0,C 180,E1 9828.76,E2 9828.76} C_VEL
LIN {X 0,Y 253.165,Z 768.781,A -85,B 0,C 180,E1 9826.169,E2 9826.169} C_VEL
LIN {X 0,Y 245.888,Z 783.38,A -85,B 0,C 180,E1 9823.165,E2 9823.165} C_VEL
LIN {X 0,Y 238.197,Z 797.674,A -85,B 0,C 180,E1 9819.455,E2 9819.455} C_VEL
LIN {X 0,Y 231.312,Z 809.761,A -85,B 0,C 180,E1 9815.459,E2 9815.459} C_VEL
LIN {X 0,Y 224.988,Z 820.583,A -85,B 0,C 180,E1 9810.865,E2 9810.865} C_VEL
LIN {X 0,Y 219.921,Z 829.206,A -85,B 0,C 180,E1 9806.092,E2 9806.092} C_VEL
